QRS_NEXT_CUT()
PTP {E1 28976.874,E2 28976.874}
PTP {X 0,Y 607.926,A -85,B 0,C 180,E1 28976.874,E2 28976.874,E3 0,E4 0,E5 0,E6 0}
QRS_SPEED_INIT()
LIN {X 0,Y 607.926,Z 799,A -85,B 0,C 180,E1 28976.874,E2 28976.874,E3 0,E4 0,E5 0,E6 0} C_VEL
LIN {X 0,Y 607.926,Z 746.583,A -85,B 0,C 180,E1 28976.874,E2 28976.874} C_VEL
LIN {X 0,Y 607.926,Z 738.171,A -85,B 0,C 180,E1 28976.874,E2 28976.874} C_VEL
LIN {X 0,Y 607.916,Z 736.195,A -85,B 0,C 180,E1 28976.715,E2 28976.715} C_VEL
LIN {X 0,Y 607.917,Z 732.197,A -85,B 0,C 180,E1 28974.904,E2 28974.904} C_VEL
LIN {X 0,Y 607.91,Z 726.378,A -85,B 0,C 180,E1 28973.104,E2 28973.104} C_VEL
LIN {X 0,Y 607.913,Z 719.011,A -85,B 0,C 180,E1 28971.392,E2 28971.392} C_VEL
LIN {X 0,Y 607.912,Z 710.203,A -85,B 0,C 180,E1 28969.768,E2 28969.768} C_VEL
LIN {X 0,Y 607.913,Z 699.301,A -85,B 0,C 180,E1 28968.132,E2 28968.132} C_VEL
LIN {X 0,Y 607.913,Z 686.828,A -85,B 0,C 180,E1 28966.59,E2 28966.59} C_VEL
LIN {X 0,Y 607.915,Z 673.153,A -85,B 0,C 180,E1 28965.181,E2 28965.181} C_VEL
LIN {X 0,Y 607.917,Z 658.405,A -85,B 0,C 180,E1 28963.91,E2 28963.91} C_VEL
LIN {X 0,Y 607.919,Z 642.683,A -85,B 0,C 180,E1 28962.779,E2 28962.779} C_VEL
LIN {X 0,Y 607.913,Z 626.024,A -85,B 0,C 180,E1 28961.79,E2 28961.79} C_VEL
LIN {X 0,Y 607.915,Z 608.442,A -85,B 0,C 180,E1 28960.944,E2 28960.944} C_VEL
LIN {X 0,Y 607.91,Z 590.522,A -85,B 0,C 180,E1 28960.27,E2 28960.27} C_VEL
LIN {X 0,Y 607.91,Z 572.648,A -85,B 0,C 180,E1 28959.768,E2 28959.768} C_VEL
LIN {X 0,Y 607.915,Z 554.05,A -85,B 0,C 180,E1 28959.417,E2 28959.417} C_VEL
LIN {X 0,Y 607.913,Z 342.093,A -85,B 0,C 180,E1 28956.75,E2 28956.75} C_VEL
LIN {X 0,Y 607.872,Z 299.576,A -85,B 0,C 180,E1 28953.695,E2 28953.695} C_VEL
LIN {X 0,Y 607.918,Z 261.354,A -85,B 0,C 180,E1 28950.867,E2 28950.867} C_VEL
LIN {X 0,Y 607.912,Z 260.757,A -85,B 0,C 180,E1 28950.65,E2 28950.65} C_VEL
LIN {X 0,Y 607.867,Z 260.764,A -85,B 0,C 180,E1 28947.546,E2 28947.546} C_VEL
LIN {X 0,Y 607.884,Z 260.759,A -85,B 0,C 180,E1 28944.273,E2 28944.273} C_VEL
LIN {X 0,Y 607.911,Z 260.765,A -85,B 0,C 180,E1 28941.196,E2 28941.196} C_VEL
LIN {X 0,Y 607.881,Z 260.759,A -85,B 0,C 180,E1 28937.975,E2 28937.975} C_VEL
LIN {X 0,Y 607.906,Z 260.759,A -85,B 0,C 180,E1 28934.855,E2 28934.855} C_VEL
LIN {X 0,Y 607.896,Z 260.762,A -85,B 0,C 180,E1 28931.691,E2 28931.691} C_VEL
LIN {X 0,Y 607.919,Z 260.754,A -85,B 0,C 180,E1 28928.441,E2 28928.441} C_VEL
LIN {X 0,Y 607.897,Z 260.762,A -85,B 0,C 180,E1 28925.168,E2 28925.168} C_VEL
LIN {X 0,Y 607.907,Z 260.758,A -85,B 0,C 180,E1 28922.091,E2 28922.091} C_VEL
LIN {X 0,Y 607.882,Z 260.759,A -85,B 0,C 180,E1 28918.92,E2 28918.92} C_VEL
LIN {X 0,Y 607.913,Z 260.765,A -85,B 0,C 180,E1 28915.736,E2 28915.736} C_VEL
LIN {X 0,Y 607.88,Z 260.759,A -85,B 0,C 180,E1 28912.638,E2 28912.638} C_VEL
LIN {X 0,Y 607.875,Z 260.763,A -85,B 0,C 180,E1 28909.407,E2 28909.407} C_VEL
LIN {X 0,Y 607.886,Z 260.76,A -85,B 0,C 180,E1 28906.435,E2 28906.435} C_VEL
LIN {X 0,Y 607.853,Z 260.764,A -85,B 0,C 180,E1 28903.315,E2 28903.315} C_VEL
LIN {X 0,Y 607.88,Z 260.763,A -85,B 0,C 180,E1 28900.385,E2 28900.385} C_VEL
LIN {X 0,Y 607.835,Z 260.767,A -85,B 0,C 180,E1 28897.278,E2 28897.278} C_VEL
LIN {X 0,Y 607.89,Z 260.966,A -85,B 0,C 180,E1 28896.257,E2 28896.257} C_VEL
LIN {X 0,Y 607.917,Z 266.861,A -85,B 0,C 180,E1 28895.759,E2 28895.759} C_VEL
LIN {X 0,Y 607.901,Z 307.026,A -85,B 0,C 180,E1 28892.688,E2 28892.688} C_VEL
LIN {X 0,Y 607.906,Z 348.222,A -85,B 0,C 180,E1 28889.624,E2 28889.624} C_VEL
LIN {X 0,Y 607.895,Z 390.467,A -85,B 0,C 180,E1 28886.559,E2 28886.559} C_VEL
LIN {X 0,Y 607.879,Z 435.108,A -85,B 0,C 180,E1 28883.39,E2 28883.39} C_VEL
LIN {X 0,Y 607.906,Z 472.483,A -85,B 0,C 180,E1 28880.797,E2 28880.797} C_VEL
LIN {X 0,Y 607.898,Z 614.271,A -85,B 0,C 180,E1 28879.072,E2 28879.072} C_VEL
LIN {X 0,Y 607.919,Z 631.005,A -85,B 0,C 180,E1 28878.69,E2 28878.69} C_VEL
LIN {X 0,Y 607.916,Z 645.866,A -85,B 0,C 180,E1 28878.185,E2 28878.185} C_VEL
LIN {X 0,Y 607.916,Z 660.472,A -85,B 0,C 180,E1 28877.51,E2 28877.51} C_VEL
LIN {X 0,Y 607.918,Z 675.006,A -85,B 0,C 180,E1 28876.64,E2 28876.64} C_VEL
LIN {X 0,Y 607.918,Z 687.294,A -85,B 0,C 180,E1 28875.718,E2 28875.718} C_VEL
LIN {X 0,Y 607.918,Z 699.759,A -85,B 0,C 180,E1 28874.548,E2 28874.548} C_VEL
LIN {X 0,Y 607.917,Z 709.872,A -85,B 0,C 180,E1 28873.372,E2 28873.372} C_VEL
LIN {X 0,Y 607.917,Z 719.257,A -85,B 0,C 180,E1 28871.99,E2 28871.99} C_VEL
LIN {X 0,Y 607.917,Z 726.624,A -85,B 0,C 180,E1 28870.597,E2 28870.597} C_VEL
LIN {X 0,Y 607.918,Z 732.436,A -85,B 0,C 180,E1 28869.091,E2 28869.091} C_VEL
LIN {X 0,Y 607.919,Z 736.408,A -85,B 0,C 180,E1 28867.57,E2 28867.57} C_VEL
LIN {X 0,Y 607.917,Z 738.54,A -85,B 0,C 180,E1 28866.032,E2 28866.032} C_VEL
LIN {X 0,Y 607.916,Z 738.894,A -85,B 0,C 180,E1 28864.476,E2 28864.476} C_VEL
LIN {X 0,Y 607.914,Z 737.56,A -85,B 0,C 180,E1 28863.004,E2 28863.004} C_VEL
LIN {X 0,Y 607.916,Z 734.271,A -85,B 0,C 180,E1 28861.437,E2 28861.437} C_VEL
LIN {X 0,Y 607.914,Z 729.539,A -85,B 0,C 180,E1 28860.002,E2 28860.002} C_VEL
LIN {X 0,Y 607.915,Z 722.969,A -85,B 0,C 180,E1 28858.577,E2 28858.577} C_VEL
LIN {X 0,Y 607.919,Z 714.179,A -85,B 0,C 180,E1 28857.13,E2 28857.13} C_VEL
LIN {X 0,Y 607.917,Z 704.536,A -85,B 0,C 180,E1 28855.887,E2 28855.887} C_VEL
LIN {X 0,Y 607.918,Z 692.695,A -85,B 0,C 180,E1 28854.666,E2 28854.666} C_VEL
LIN {X 0,Y 607.918,Z 680.197,A -85,B 0,C 180,E1 28853.637,E2 28853.637} C_VEL
LIN {X 0,Y 607.906,Z 665.842,A -85,B 0,C 180,E1 28852.694,E2 28852.694} C_VEL
LIN {X 0,Y 607.904,Z 651.24,A -85,B 0,C 180,E1 28851.953,E2 28851.953} C_VEL
LIN {X 0,Y 607.917,Z 635.281,A -85,B 0,C 180,E1 28851.348,E2 28851.348} C_VEL
LIN {X 0,Y 607.896,Z 619.814,A -85,B 0,C 180,E1 28850.941,E2 28850.941} C_VEL
LIN {X 0,Y 607.871,Z 600.343,A -85,B 0,C 180,E1 28850.652,E2 28850.652} C_VEL
LIN {X 0,Y 607.901,Z 472.16,A -85,B 0,C 180,E1 28849.1,E2 28849.1} C_VEL
LIN {X 0,Y 607.844,Z 432.037,A -85,B 0,C 180,E1 28846.303,E2 28846.303} C_VEL
LIN {X 0,Y 607.882,Z 388.77,A -85,B 0,C 180,E1 28843.228,E2 28843.228} C_VEL
LIN {X 0,Y 607.899,Z 347.838,A -85,B 0,C 180,E1 28840.257,E2 28840.257} C_VEL
LIN {X 0,Y 607.913,Z 306.577,A -85,B 0,C 180,E1 28837.189,E2 28837.189} C_VEL
LIN {X 0,Y 607.919,Z 265.74,A -85,B 0,C 180,E1 28834.064,E2 28834.064} C_VEL
LIN {X 0,Y 607.913,Z 260.992,A -85,B 0,C 180,E1 28833.661,E2 28833.661} C_VEL
LIN {X 0,Y 607.864,Z 260.761,A -85,B 0,C 180,E1 28830.657,E2 28830.657} C_VEL
LIN {X 0,Y 607.915,Z 260.761,A -85,B 0,C 180,E1 28827.566,E2 28827.566} C_VEL
LIN {X 0,Y 607.864,Z 260.761,A -85,B 0,C 180,E1 28824.489,E2 28824.489} C_VEL
LIN {X 0,Y 607.915,Z 260.758,A -85,B 0,C 180,E1 28821.315,E2 28821.315} C_VEL
LIN {X 0,Y 607.871,Z 260.762,A -85,B 0,C 180,E1 28818.212,E2 28818.212} C_VEL
LIN {X 0,Y 607.895,Z 260.757,A -85,B 0,C 180,E1 28814.966,E2 28814.966} C_VEL
LIN {X 0,Y 607.892,Z 260.764,A -85,B 0,C 180,E1 28811.865,E2 28811.865} C_VEL
LIN {X 0,Y 607.874,Z 260.759,A -85,B 0,C 180,E1 28808.609,E2 28808.609} C_VEL
LIN {X 0,Y 607.911,Z 260.766,A -85,B 0,C 180,E1 28805.569,E2 28805.569} C_VEL
LIN {X 0,Y 607.871,Z 260.759,A -85,B 0,C 180,E1 28802.451,E2 28802.451} C_VEL
LIN {X 0,Y 607.914,Z 260.762,A -85,B 0,C 180,E1 28799.341,E2 28799.341} C_VEL
LIN {X 0,Y 607.87,Z 260.76,A -85,B 0,C 180,E1 28796.228,E2 28796.228} C_VEL
LIN {X 0,Y 607.911,Z 260.759,A -85,B 0,C 180,E1 28793.104,E2 28793.104} C_VEL
LIN {X 0,Y 607.872,Z 260.761,A -85,B 0,C 180,E1 28790.055,E2 28790.055} C_VEL
LIN {X 0,Y 607.915,Z 260.756,A -85,B 0,C 180,E1 28786.818,E2 28786.818} C_VEL
LIN {X 0,Y 607.89,Z 260.763,A -85,B 0,C 180,E1 28783.665,E2 28783.665} C_VEL
LIN {X 0,Y 607.882,Z 260.758,A -85,B 0,C 180,E1 28780.395,E2 28780.395} C_VEL
LIN {X 0,Y 607.916,Z 260.764,A -85,B 0,C 180,E1 28777.263,E2 28777.263} C_VEL
LIN {X 0,Y 607.875,Z 260.759,A -85,B 0,C 180,E1 28774.119,E2 28774.119} C_VEL
LIN {X 0,Y 607.911,Z 260.76,A -85,B 0,C 180,E1 28770.975,E2 28770.975} C_VEL
LIN {X 0,Y 607.875,Z 260.76,A -85,B 0,C 180,E1 28767.894,E2 28767.894} C_VEL
LIN {X 0,Y 607.914,Z 260.757,A -85,B 0,C 180,E1 28764.739,E2 28764.739} C_VEL
LIN {X 0,Y 607.88,Z 260.761,A -85,B 0,C 180,E1 28761.677,E2 28761.677} C_VEL
LIN {X 0,Y 607.905,Z 260.756,A -85,B 0,C 180,E1 28758.447,E2 28758.447} C_VEL
LIN {X 0,Y 607.908,Z 260.764,A -85,B 0,C 180,E1 28755.255,E2 28755.255} C_VEL
LIN {X 0,Y 607.882,Z 260.758,A -85,B 0,C 180,E1 28752.022,E2 28752.022} C_VEL
LIN {X 0,Y 607.912,Z 260.762,A -85,B 0,C 180,E1 28748.922,E2 28748.922} C_VEL
LIN {X 0,Y 607.878,Z 260.757,A -85,B 0,C 180,E1 28745.816,E2 28745.816} C_VEL
LIN {X 0,Y 607.909,Z 260.758,A -85,B 0,C 180,E1 28742.758,E2 28742.758} C_VEL
LIN {X 0,Y 607.901,Z 261.045,A -85,B 0,C 180,E1 28741.19,E2 28741.19} C_VEL
LIN {X 0,Y 607.917,Z 270.434,A -85,B 0,C 180,E1 28740.544,E2 28740.544} C_VEL
LIN {X 0,Y 607.883,Z 315.134,A -85,B 0,C 180,E1 28737.7,E2 28737.7} C_VEL
LIN {X 0,Y 607.916,Z 528.002,A -85,B 0,C 180,E1 28734.938,E2 28734.938} C_VEL
LIN {X 0,Y 607.917,Z 577.773,A -85,B 0,C 180,E1 28734.278,E2 28734.278} C_VEL
LIN {X 0,Y 607.906,Z 597.727,A -85,B 0,C 180,E1 28733.84,E2 28733.84} C_VEL
LIN {X 0,Y 607.911,Z 617.08,A -85,B 0,C 180,E1 28733.248,E2 28733.248} C_VEL
LIN {X 0,Y 607.916,Z 636.502,A -85,B 0,C 180,E1 28732.482,E2 28732.482} C_VEL
LIN {X 0,Y 607.919,Z 655.181,A -85,B 0,C 180,E1 28731.566,E2 28731.566} C_VEL
LIN {X 0,Y 607.917,Z 673.777,A -85,B 0,C 180,E1 28730.456,E2 28730.456} C_VEL
LIN {X 0,Y 607.915,Z 691.264,A -85,B 0,C 180,E1 28729.204,E2 28729.204} C_VEL
LIN {X 0,Y 607.914,Z 707.171,A -85,B 0,C 180,E1 28727.862,E2 28727.862} C_VEL
LIN {X 0,Y 607.917,Z 721.68,A -85,B 0,C 180,E1 28726.432,E2 28726.432} C_VEL
LIN {X 0,Y 607.909,Z 735.27,A -85,B 0,C 180,E1 28724.866,E2 28724.866} C_VEL
LIN {X 0,Y 607.906,Z 747.75,A -85,B 0,C 180,E1 28723.171,E2 28723.171} C_VEL
LIN {X 0,Y 607.905,Z 758.257,A -85,B 0,C 180,E1 28721.478,E2 28721.478} C_VEL
LIN {X 0,Y 607.912,Z 767.565,A -85,B 0,C 180,E1 28719.657,E2 28719.657} C_VEL
LIN {X 0,Y 607.914,Z 774.977,A -85,B 0,C 180,E1 28717.845,E2 28717.845} C_VEL
LIN {X 0,Y 607.918,Z 780.991,A -85,B 0,C 180,E1 28715.946,E2 28715.946} C_VEL
LIN {X 0,Y 607.916,Z 785.294,A -85,B 0,C 180,E1 28714.054,E2 28714.054} C_VEL
LIN {X 0,Y 607.914,Z 788.04,A -85,B 0,C 180,E1 28712.073,E2 28712.073} C_VEL
LIN {X 0,Y 607.912,Z 788.984,A -85,B 0,C 180,E1 28710.093,E2 28710.093} C_VEL
LIN {X 0,Y 607.91,Z 788.239,A -85,B 0,C 180,E1 28708.208,E2 28708.208} C_VEL
LIN {X 0,Y 607.915,Z 785.764,A -85,B 0,C 180,E1 28706.227,E2 28706.227} C_VEL
LIN {X 0,Y 607.914,Z 781.492,A -85,B 0,C 180,E1 28704.241,E2 28704.241} C_VEL
LIN {X 0,Y 607.913,Z 776.031,A -85,B 0,C 180,E1 28702.438,E2 28702.438} C_VEL
LIN {X 0,Y 607.911,Z 768.837,A -85,B 0,C 180,E1 28700.628,E2 28700.628} C_VEL
LIN {X 0,Y 607.909,Z 760.319,A -85,B 0,C 180,E1 28698.904,E2 28698.904} C_VEL
LIN {X 0,Y 607.914,Z 749.368,A -85,B 0,C 180,E1 28697.074,E2 28697.074} C_VEL
LIN {X 0,Y 607.911,Z 737.579,A -85,B 0,C 180,E1 28695.424,E2 28695.424} C_VEL
LIN {X 0,Y 607.918,Z 724.302,A -85,B 0,C 180,E1 28693.846,E2 28693.846} C_VEL
LIN {X 0,Y 607.916,Z 709.355,A -85,B 0,C 180,E1 28692.334,E2 28692.334} C_VEL
LIN {X 0,Y 607.914,Z 692.556,A -85,B 0,C 180,E1 28690.894,E2 28690.894} C_VEL
LIN {X 0,Y 607.916,Z 674.521,A -85,B 0,C 180,E1 28689.592,E2 28689.592} C_VEL
LIN {X 0,Y 607.919,Z 656.038,A -85,B 0,C 180,E1 28688.482,E2 28688.482} C_VEL
LIN {X 0,Y 607.916,Z 637.586,A -85,B 0,C 180,E1 28687.568,E2 28687.568} C_VEL
LIN {X 0,Y 607.909,Z 618.324,A -85,B 0,C 180,E1 28686.795,E2 28686.795} C_VEL
LIN {X 0,Y 607.906,Z 598.676,A -85,B 0,C 180,E1 28686.184,E2 28686.184} C_VEL
LIN {X 0,Y 607.918,Z 578.992,A -85,B 0,C 180,E1 28685.746,E2 28685.746} C_VEL
LIN {X 0,Y 607.91,Z 541.04,A -85,B 0,C 180,E1 28685.228,E2 28685.228} C_VEL
LIN {X 0,Y 607.883,Z 316.158,A -85,B 0,C 180,E1 28682.324,E2 28682.324} C_VEL
LIN {X 0,Y 607.885,Z 313.372,A -85,B 0,C 180,E1 28682.196,E2 28682.196} C_VEL
LIN {X 0,Y 607.918,Z 267.016,A -85,B 0,C 180,E1 28679.235,E2 28679.235} C_VEL
LIN {X 0,Y 607.903,Z 261.097,A -85,B 0,C 180,E1 28678.822,E2 28678.822} C_VEL
LIN {X 0,Y 607.884,Z 260.755,A -85,B 0,C 180,E1 28678.073,E2 28678.073} C_VEL
LIN {X 0,Y 607.904,Z 260.764,A -85,B 0,C 180,E1 28674.83,E2 28674.83} C_VEL
LIN {X 0,Y 607.919,Z 260.756,A -85,B 0,C 180,E1 28671.559,E2 28671.559} C_VEL
LIN {X 0,Y 607.873,Z 260.761,A -85,B 0,C 180,E1 28668.354,E2 28668.354} C_VEL
LIN {X 0,Y 607.913,Z 260.76,A -85,B 0,C 180,E1 28665.255,E2 28665.255} C_VEL
LIN {X 0,Y 607.868,Z 260.76,A -85,B 0,C 180,E1 28662.152,E2 28662.152} C_VEL
LIN {X 0,Y 607.917,Z 260.764,A -85,B 0,C 180,E1 28659.045,E2 28659.045} C_VEL
LIN {X 0,Y 607.867,Z 260.76,A -85,B 0,C 180,E1 28655.959,E2 28655.959} C_VEL
LIN {X 0,Y 607.894,Z 260.765,A -85,B 0,C 180,E1 28652.761,E2 28652.761} C_VEL
LIN {X 0,Y 607.875,Z 260.757,A -85,B 0,C 180,E1 28649.717,E2 28649.717} C_VEL
LIN {X 0,Y 607.917,Z 261.074,A -85,B 0,C 180,E1 28649.079,E2 28649.079} C_VEL
LIN {X 0,Y 607.882,Z 296.062,A -85,B 0,C 180,E1 28646.471,E2 28646.471} C_VEL
LIN {X 0,Y 607.915,Z 339.268,A -85,B 0,C 180,E1 28643.352,E2 28643.352} C_VEL
LIN {X 0,Y 607.913,Z 342.484,A -85,B 0,C 180,E1 28643.147,E2 28643.147} C_VEL
LIN {X 0,Y 607.914,Z 559.808,A -85,B 0,C 180,E1 28640.407,E2 28640.407} C_VEL
LIN {X 0,Y 607.914,Z 579.217,A -85,B 0,C 180,E1 28639.98,E2 28639.98} C_VEL
LIN {X 0,Y 607.914,Z 597.431,A -85,B 0,C 180,E1 28639.404,E2 28639.404} C_VEL
LIN {X 0,Y 607.915,Z 615.767,A -85,B 0,C 180,E1 28638.639,E2 28638.639} C_VEL
LIN {X 0,Y 607.918,Z 633.298,A -85,B 0,C 180,E1 28637.714,E2 28637.714} C_VEL
LIN {X 0,Y 607.915,Z 650.04,A -85,B 0,C 180,E1 28636.629,E2 28636.629} C_VEL
LIN {X 0,Y 607.917,Z 665.659,A -85,B 0,C 180,E1 28635.404,E2 28635.404} C_VEL
LIN {X 0,Y 607.915,Z 679.684,A -85,B 0,C 180,E1 28634.088,E2 28634.088} C_VEL
LIN {X 0,Y 607.915,Z 692.662,A -85,B 0,C 180,E1 28632.635,E2 28632.635} C_VEL
LIN {X 0,Y 607.917,Z 704.133,A -85,B 0,C 180,E1 28631.095,E2 28631.095} C_VEL
LIN {X 0,Y 607.911,Z 714.103,A -85,B 0,C 180,E1 28629.466,E2 28629.466} C_VEL
LIN {X 0,Y 607.912,Z 722.146,A -85,B 0,C 180,E1 28627.846,E2 28627.846} C_VEL
LIN {X 0,Y 607.91,Z 728.788,A -85,B 0,C 180,E1 28626.137,E2 28626.137} C_VEL
LIN {X 0,Y 607.905,Z 733.703,A -85,B 0,C 180,E1 28624.433,E2 28624.433} C_VEL
LIN {X 0,Y 607.908,Z 737.107,A -85,B 0,C 180,E1 28622.639,E2 28622.639} C_VEL
LIN {X 0,Y 607.917,Z 738.818,A -85,B 0,C 180,E1 28620.754,E2 28620.754} C_VEL
LIN {X 0,Y 607.915,Z 738.727,A -85,B 0,C 180,E1 28618.963,E2 28618.963} C_VEL
LIN {X 0,Y 607.912,Z 736.955,A -85,B 0,C 180,E1 28617.171,E2 28617.171} C_VEL
LIN {X 0,Y 607.916,Z 736.195,A -85,B 0,C 180,E1 28616.715,E2 28616.715} C_VEL
LIN {X 0,Y 606.897,Z 734.89,A -85,B 0,C 180,E1 28615.999,E2 28615.999} C_VEL
LIN {X 0,Y 601.771,Z 731.347,A -85,B 0,C 180,E1 28614.518,E2 28614.518} C_VEL
LIN {X 0,Y 600.007,Z 728.896,A -85,B 0,C 180,E1 28613.716,E2 28613.716} C_VEL
LIN {X 0,Y 599.918,Z 728.211,A -85,B 0,C 180,E1 28613.514,E2 28613.514} C_VEL
LIN {X 0,Y 599.921,Z 721.302,A -85,B 0,C 180,E1 28611.759,E2 28611.759} C_VEL
LIN {X 0,Y 599.942,Z 712.5,A -85,B 0,C 180,E1 28610.018,E2 28610.018} C_VEL
LIN {X 0,Y 599.964,Z 702.139,A -85,B 0,C 180,E1 28608.366,E2 28608.366} C_VEL
LIN {X 0,Y 600.005,Z 690.217,A -85,B 0,C 180,E1 28606.803,E2 28606.803} C_VEL
LIN {X 0,Y 600.044,Z 676.686,A -85,B 0,C 180,E1 28605.328,E2 28605.328} C_VEL
LIN {X 0,Y 600.096,Z 662.408,A -85,B 0,C 180,E1 28604.025,E2 28604.025} C_VEL
LIN {X 0,Y 600.153,Z 647.039,A -85,B 0,C 180,E1 28602.849,E2 28602.849} C_VEL
LIN {X 0,Y 600.218,Z 630.474,A -85,B 0,C 180,E1 28601.799,E2 28601.799} C_VEL
LIN {X 0,Y 600.273,Z 614.032,A -85,B 0,C 180,E1 28600.945,E2 28600.945} C_VEL
LIN {X 0,Y 600.329,Z 595.811,A -85,B 0,C 180,E1 28600.193,E2 28600.193} C_VEL
LIN {X 0,Y 600.38,Z 576.816,A -85,B 0,C 180,E1 28599.606,E2 28599.606} C_VEL
LIN {X 0,Y 600.415,Z 557.875,A -85,B 0,C 180,E1 28599.205,E2 28599.205} C_VEL
LIN {X 0,Y 600.429,Z 342.582,A -85,B 0,C 180,E1 28596.459,E2 28596.459} C_VEL
LIN {X 0,Y 600.422,Z 301.598,A -85,B 0,C 180,E1 28593.494,E2 28593.494} C_VEL
LIN {X 0,Y 600.567,Z 263.941,A -85,B 0,C 180,E1 28590.68,E2 28590.68} C_VEL
LIN {X 0,Y 599.967,Z 261.874,A -85,B 0,C 180,E1 28590.442,E2 28590.442} C_VEL
LIN {X 0,Y 599.936,Z 261.754,A -85,B 0,C 180,E1 28587.43,E2 28587.43} C_VEL
LIN {X 0,Y 599.94,Z 261.748,A -85,B 0,C 180,E1 28584.198,E2 28584.198} C_VEL
LIN {X 0,Y 599.974,Z 261.753,A -85,B 0,C 180,E1 28581.077,E2 28581.077} C_VEL
LIN {X 0,Y 599.942,Z 261.749,A -85,B 0,C 180,E1 28577.871,E2 28577.871} C_VEL
LIN {X 0,Y 599.97,Z 261.746,A -85,B 0,C 180,E1 28574.691,E2 28574.691} C_VEL
LIN {X 0,Y 599.975,Z 261.753,A -85,B 0,C 180,E1 28571.415,E2 28571.415} C_VEL
LIN {X 0,Y 599.961,Z 261.746,A -85,B 0,C 180,E1 28568.13,E2 28568.13} C_VEL
LIN {X 0,Y 599.953,Z 261.749,A -85,B 0,C 180,E1 28564.981,E2 28564.981} C_VEL
LIN {X 0,Y 599.97,Z 261.751,A -85,B 0,C 180,E1 28561.778,E2 28561.778} C_VEL
LIN {X 0,Y 599.958,Z 261.745,A -85,B 0,C 180,E1 28558.564,E2 28558.564} C_VEL
LIN {X 0,Y 599.942,Z 261.75,A -85,B 0,C 180,E1 28555.256,E2 28555.256} C_VEL
LIN {X 0,Y 599.977,Z 261.748,A -85,B 0,C 180,E1 28552.092,E2 28552.092} C_VEL
LIN {X 0,Y 599.922,Z 261.751,A -85,B 0,C 180,E1 28548.966,E2 28548.966} C_VEL
LIN {X 0,Y 599.972,Z 261.753,A -85,B 0,C 180,E1 28545.862,E2 28545.862} C_VEL
LIN {X 0,Y 599.911,Z 261.752,A -85,B 0,C 180,E1 28542.834,E2 28542.834} C_VEL
LIN {X 0,Y 599.922,Z 261.755,A -85,B 0,C 180,E1 28539.595,E2 28539.595} C_VEL
LIN {X 0,Y 599.905,Z 261.757,A -85,B 0,C 180,E1 28536.701,E2 28536.701} C_VEL
LIN {X 0,Y 599.985,Z 262.18,A -85,B 0,C 180,E1 28536.508,E2 28536.508} C_VEL
LIN {X 0,Y 600.494,Z 265.704,A -85,B 0,C 180,E1 28536.214,E2 28536.214} C_VEL
LIN {X 0,Y 600.557,Z 294.621,A -85,B 0,C 180,E1 28534.011,E2 28534.011} C_VEL
LIN {X 0,Y 600.422,Z 335.458,A -85,B 0,C 180,E1 28530.907,E2 28530.907} C_VEL
LIN {X 0,Y 600.294,Z 376.693,A -85,B 0,C 180,E1 28527.853,E2 28527.853} C_VEL
LIN {X 0,Y 600.211,Z 418.923,A -85,B 0,C 180,E1 28524.792,E2 28524.792} C_VEL
LIN {X 0,Y 600.106,Z 464.253,A -85,B 0,C 180,E1 28521.57,E2 28521.57} C_VEL
LIN {X 0,Y 600.166,Z 472.786,A -85,B 0,C 180,E1 28521.001,E2 28521.001} C_VEL
LIN {X 0,Y 600.135,Z 615.243,A -85,B 0,C 180,E1 28519.241,E2 28519.241} C_VEL
LIN {X 0,Y 600.133,Z 632.155,A -85,B 0,C 180,E1 28518.84,E2 28518.84} C_VEL
LIN {X 0,Y 600.099,Z 646.835,A -85,B 0,C 180,E1 28518.322,E2 28518.322} C_VEL
LIN {X 0,Y 600.061,Z 662.094,A -85,B 0,C 180,E1 28517.589,E2 28517.589} C_VEL
LIN {X 0,Y 600.029,Z 676.504,A -85,B 0,C 180,E1 28516.695,E2 28516.695} C_VEL
LIN {X 0,Y 599.994,Z 689.443,A -85,B 0,C 180,E1 28515.674,E2 28515.674} C_VEL
LIN {X 0,Y 599.968,Z 701.086,A -85,B 0,C 180,E1 28514.537,E2 28514.537} C_VEL
LIN {X 0,Y 599.945,Z 711.629,A -85,B 0,C 180,E1 28513.244,E2 28513.244} C_VEL
LIN {X 0,Y 599.933,Z 720.689,A -85,B 0,C 180,E1 28511.842,E2 28511.842} C_VEL
LIN {X 0,Y 599.919,Z 727.663,A -85,B 0,C 180,E1 28510.429,E2 28510.429} C_VEL
LIN {X 0,Y 599.915,Z 733.208,A -85,B 0,C 180,E1 28508.901,E2 28508.901} C_VEL
LIN {X 0,Y 599.914,Z 736.863,A -85,B 0,C 180,E1 28507.358,E2 28507.358} C_VEL
LIN {X 0,Y 599.916,Z 738.786,A -85,B 0,C 180,E1 28505.692,E2 28505.692} C_VEL
LIN {X 0,Y 599.914,Z 738.746,A -85,B 0,C 180,E1 28504.16,E2 28504.16} C_VEL
LIN {X 0,Y 599.915,Z 736.787,A -85,B 0,C 180,E1 28502.507,E2 28502.507} C_VEL
LIN {X 0,Y 599.915,Z 733.146,A -85,B 0,C 180,E1 28500.989,E2 28500.989} C_VEL
LIN {X 0,Y 599.922,Z 727.529,A -85,B 0,C 180,E1 28499.449,E2 28499.449} C_VEL
LIN {X 0,Y 599.931,Z 720.468,A -85,B 0,C 180,E1 28498.029,E2 28498.029} C_VEL
LIN {X 0,Y 599.944,Z 711.414,A -85,B 0,C 180,E1 28496.637,E2 28496.637} C_VEL
LIN {X 0,Y 599.969,Z 701.066,A -85,B 0,C 180,E1 28495.371,E2 28495.371} C_VEL
LIN {X 0,Y 599.994,Z 689.078,A -85,B 0,C 180,E1 28494.204,E2 28494.204} C_VEL
LIN {X 0,Y 600.031,Z 676.113,A -85,B 0,C 180,E1 28493.189,E2 28493.189} C_VEL
LIN {X 0,Y 600.058,Z 661.752,A -85,B 0,C 180,E1 28492.302,E2 28492.302} C_VEL
LIN {X 0,Y 600.086,Z 647.798,A -85,B 0,C 180,E1 28491.629,E2 28491.629} C_VEL
LIN {X 0,Y 600.132,Z 632.099,A -85,B 0,C 180,E1 28491.069,E2 28491.069} C_VEL
LIN {X 0,Y 600.123,Z 615.12,A -85,B 0,C 180,E1 28490.667,E2 28490.667} C_VEL
LIN {X 0,Y 600.114,Z 472.239,A -85,B 0,C 180,E1 28488.893,E2 28488.893} C_VEL
LIN {X 0,Y 600.13,Z 431.749,A -85,B 0,C 180,E1 28486.034,E2 28486.034} C_VEL
LIN {X 0,Y 600.243,Z 387.092,A -85,B 0,C 180,E1 28482.815,E2 28482.815} C_VEL
LIN {X 0,Y 600.39,Z 347.187,A -85,B 0,C 180,E1 28479.879,E2 28479.879} C_VEL
LIN {X 0,Y 600.534,Z 305.133,A -85,B 0,C 180,E1 28476.707,E2 28476.707} C_VEL
LIN {X 0,Y 600.531,Z 270.72,A -85,B 0,C 180,E1 28474.074,E2 28474.074} C_VEL
LIN {X 0,Y 600.134,Z 262.619,A -85,B 0,C 180,E1 28473.468,E2 28473.468} C_VEL
LIN {X 0,Y 599.97,Z 261.765,A -85,B 0,C 180,E1 28473.291,E2 28473.291} C_VEL
LIN {X 0,Y 599.935,Z 261.753,A -85,B 0,C 180,E1 28470.22,E2 28470.22} C_VEL
LIN {X 0,Y 599.94,Z 261.748,A -85,B 0,C 180,E1 28466.925,E2 28466.925} C_VEL
LIN {X 0,Y 599.972,Z 261.754,A -85,B 0,C 180,E1 28463.785,E2 28463.785} C_VEL
LIN {X 0,Y 599.929,Z 261.749,A -85,B 0,C 180,E1 28460.589,E2 28460.589} C_VEL
LIN {X 0,Y 599.976,Z 261.75,A -85,B 0,C 180,E1 28457.456,E2 28457.456} C_VEL
LIN {X 0,Y 599.928,Z 261.75,A -85,B 0,C 180,E1 28454.379,E2 28454.379} C_VEL
LIN {X 0,Y 599.975,Z 261.747,A -85,B 0,C 180,E1 28451.244,E2 28451.244} C_VEL
LIN {X 0,Y 599.933,Z 261.751,A -85,B 0,C 180,E1 28448.135,E2 28448.135} C_VEL
LIN {X 0,Y 599.959,Z 261.746,A -85,B 0,C 180,E1 28444.876,E2 28444.876} C_VEL
LIN {X 0,Y 599.959,Z 261.753,A -85,B 0,C 180,E1 28441.719,E2 28441.719} C_VEL
LIN {X 0,Y 599.935,Z 261.748,A -85,B 0,C 180,E1 28438.472,E2 28438.472} C_VEL
LIN {X 0,Y 599.975,Z 261.751,A -85,B 0,C 180,E1 28435.316,E2 28435.316} C_VEL
LIN {X 0,Y 599.931,Z 261.75,A -85,B 0,C 180,E1 28432.146,E2 28432.146} C_VEL
LIN {X 0,Y 599.976,Z 261.746,A -85,B 0,C 180,E1 28428.951,E2 28428.951} C_VEL
LIN {X 0,Y 599.942,Z 261.751,A -85,B 0,C 180,E1 28425.819,E2 28425.819} C_VEL
LIN {X 0,Y 599.952,Z 261.746,A -85,B 0,C 180,E1 28422.544,E2 28422.544} C_VEL
LIN {X 0,Y 599.978,Z 261.753,A -85,B 0,C 180,E1 28419.311,E2 28419.311} C_VEL
LIN {X 0,Y 599.935,Z 261.749,A -85,B 0,C 180,E1 28416.11,E2 28416.11} C_VEL
LIN {X 0,Y 599.973,Z 261.748,A -85,B 0,C 180,E1 28412.938,E2 28412.938} C_VEL
LIN {X 0,Y 599.94,Z 261.75,A -85,B 0,C 180,E1 28409.781,E2 28409.781} C_VEL
LIN {X 0,Y 599.969,Z 261.745,A -85,B 0,C 180,E1 28406.522,E2 28406.522} C_VEL
LIN {X 0,Y 599.975,Z 261.754,A -85,B 0,C 180,E1 28403.254,E2 28403.254} C_VEL
LIN {X 0,Y 599.94,Z 261.748,A -85,B 0,C 180,E1 28400.05,E2 28400.05} C_VEL
LIN {X 0,Y 599.972,Z 261.75,A -85,B 0,C 180,E1 28396.901,E2 28396.901} C_VEL
LIN {X 0,Y 599.939,Z 261.749,A -85,B 0,C 180,E1 28393.758,E2 28393.758} C_VEL
LIN {X 0,Y 599.974,Z 261.746,A -85,B 0,C 180,E1 28390.535,E2 28390.535} C_VEL
LIN {X 0,Y 599.954,Z 261.753,A -85,B 0,C 180,E1 28387.344,E2 28387.344} C_VEL
LIN {X 0,Y 599.951,Z 261.748,A -85,B 0,C 180,E1 28384.052,E2 28384.052} C_VEL
LIN {X 0,Y 599.976,Z 261.995,A -85,B 0,C 180,E1 28381.589,E2 28381.589} C_VEL
LIN {X 0,Y 600.75,Z 265.362,A -85,B 0,C 180,E1 28381.282,E2 28381.282} C_VEL
LIN {X 0,Y 600.583,Z 311.765,A -85,B 0,C 180,E1 28378.275,E2 28378.275} C_VEL
LIN {X 0,Y 600.704,Z 316.046,A -85,B 0,C 180,E1 28378.038,E2 28378.038} C_VEL
LIN {X 0,Y 600.667,Z 519.783,A -85,B 0,C 180,E1 28375.367,E2 28375.367} C_VEL
LIN {X 0,Y 600.61,Z 578.292,A -85,B 0,C 180,E1 28374.583,E2 28374.583} C_VEL
LIN {X 0,Y 600.557,Z 598.764,A -85,B 0,C 180,E1 28374.124,E2 28374.124} C_VEL
LIN {X 0,Y 600.499,Z 617.817,A -85,B 0,C 180,E1 28373.526,E2 28373.526} C_VEL
LIN {X 0,Y 600.425,Z 637.639,A -85,B 0,C 180,E1 28372.725,E2 28372.725} C_VEL
LIN {X 0,Y 600.349,Z 656.078,A -85,B 0,C 180,E1 28371.8,E2 28371.8} C_VEL
LIN {X 0,Y 600.277,Z 674.551,A -85,B 0,C 180,E1 28370.677,E2 28370.677} C_VEL
LIN {X 0,Y 600.197,Z 692.585,A -85,B 0,C 180,E1 28369.359,E2 28369.359} C_VEL
LIN {X 0,Y 600.123,Z 709.379,A -85,B 0,C 180,E1 28367.901,E2 28367.901} C_VEL
LIN {X 0,Y 600.064,Z 724.878,A -85,B 0,C 180,E1 28366.309,E2 28366.309} C_VEL
LIN {X 0,Y 600.007,Z 738.373,A -85,B 0,C 180,E1 28364.671,E2 28364.671} C_VEL
LIN {X 0,Y 599.972,Z 750.023,A -85,B 0,C 180,E1 28363,E2 28363} C_VEL
LIN {X 0,Y 599.945,Z 760.331,A -85,B 0,C 180,E1 28361.243,E2 28361.243} C_VEL
LIN {X 0,Y 599.925,Z 769.36,A -85,B 0,C 180,E1 28359.373,E2 28359.373} C_VEL
LIN {X 0,Y 599.92,Z 776.383,A -85,B 0,C 180,E1 28357.565,E2 28357.565} C_VEL
LIN {X 0,Y 599.913,Z 782.004,A -85,B 0,C 180,E1 28355.642,E2 28355.642} C_VEL
LIN {X 0,Y 599.912,Z 785.926,A -85,B 0,C 180,E1 28353.726,E2 28353.726} C_VEL
LIN {X 0,Y 599.906,Z 788.307,A -85,B 0,C 180,E1 28351.718,E2 28351.718} C_VEL
LIN {X 0,Y 599.907,Z 788.962,A -85,B 0,C 180,E1 28349.808,E2 28349.808} C_VEL
LIN {X 0,Y 599.91,Z 787.949,A -85,B 0,C 180,E1 28347.802,E2 28347.802} C_VEL
LIN {X 0,Y 599.909,Z 785.133,A -85,B 0,C 180,E1 28345.794,E2 28345.794} C_VEL
LIN {X 0,Y 599.919,Z 780.733,A -85,B 0,C 180,E1 28343.876,E2 28343.876} C_VEL
LIN {X 0,Y 599.923,Z 774.616,A -85,B 0,C 180,E1 28341.951,E2 28341.951} C_VEL
LIN {X 0,Y 599.934,Z 766.799,A -85,B 0,C 180,E1 28340.053,E2 28340.053} C_VEL
LIN {X 0,Y 599.943,Z 757.711,A -85,B 0,C 180,E1 28338.268,E2 28338.268} C_VEL
LIN {X 0,Y 599.974,Z 746.81,A -85,B 0,C 180,E1 28336.507,E2 28336.507} C_VEL
LIN {X 0,Y 600.019,Z 734.479,A -85,B 0,C 180,E1 28334.833,E2 28334.833} C_VEL
LIN {X 0,Y 600.065,Z 720.733,A -85,B 0,C 180,E1 28333.245,E2 28333.245} C_VEL
LIN {X 0,Y 600.133,Z 705.441,A -85,B 0,C 180,E1 28331.741,E2 28331.741} C_VEL
LIN {X 0,Y 600.207,Z 688.595,A -85,B 0,C 180,E1 28330.335,E2 28330.335} C_VEL
LIN {X 0,Y 600.29,Z 671.337,A -85,B 0,C 180,E1 28329.117,E2 28329.117} C_VEL
LIN {X 0,Y 600.374,Z 653.234,A -85,B 0,C 180,E1 28328.044,E2 28328.044} C_VEL
LIN {X 0,Y 600.442,Z 634.219,A -85,B 0,C 180,E1 28327.118,E2 28327.118} C_VEL
LIN {X 0,Y 600.507,Z 614.815,A -85,B 0,C 180,E1 28326.368,E2 28326.368} C_VEL
LIN {X 0,Y 600.564,Z 594.781,A -85,B 0,C 180,E1 28325.776,E2 28325.776} C_VEL
LIN {X 0,Y 600.619,Z 574.279,A -85,B 0,C 180,E1 28325.354,E2 28325.354} C_VEL
LIN {X 0,Y 600.788,Z 328.828,A -85,B 0,C 180,E1 28322.137,E2 28322.137} C_VEL
LIN {X 0,Y 600.615,Z 315.45,A -85,B 0,C 180,E1 28321.946,E2 28321.946} C_VEL
LIN {X 0,Y 600.741,Z 269.622,A -85,B 0,C 180,E1 28318.998,E2 28318.998} C_VEL
LIN {X 0,Y 600.68,Z 264.235,A -85,B 0,C 180,E1 28318.639,E2 28318.639} C_VEL
LIN {X 0,Y 599.96,Z 261.887,A -85,B 0,C 180,E1 28318.386,E2 28318.386} C_VEL
LIN {X 0,Y 599.971,Z 261.752,A -85,B 0,C 180,E1 28315.244,E2 28315.244} C_VEL
LIN {X 0,Y 599.936,Z 261.749,A -85,B 0,C 180,E1 28312.17,E2 28312.17} C_VEL
LIN {X 0,Y 599.977,Z 261.754,A -85,B 0,C 180,E1 28308.958,E2 28308.958} C_VEL
LIN {X 0,Y 599.952,Z 261.747,A -85,B 0,C 180,E1 28305.776,E2 28305.776} C_VEL
LIN {X 0,Y 599.94,Z 261.752,A -85,B 0,C 180,E1 28302.554,E2 28302.554} C_VEL
LIN {X 0,Y 599.979,Z 261.747,A -85,B 0,C 180,E1 28299.415,E2 28299.415} C_VEL
LIN {X 0,Y 599.925,Z 261.751,A -85,B 0,C 180,E1 28296.229,E2 28296.229} C_VEL
LIN {X 0,Y 599.976,Z 261.752,A -85,B 0,C 180,E1 28293.135,E2 28293.135} C_VEL
LIN {X 0,Y 599.919,Z 261.744,A -85,B 0,C 180,E1 28290.11,E2 28290.11} C_VEL
LIN {X 0,Y 600.003,Z 262.027,A -85,B 0,C 180,E1 28289.43,E2 28289.43} C_VEL
LIN {X 0,Y 600.581,Z 265.108,A -85,B 0,C 180,E1 28289.141,E2 28289.141} C_VEL
LIN {X 0,Y 600.412,Z 305.124,A -85,B 0,C 180,E1 28286.156,E2 28286.156} C_VEL
LIN {X 0,Y 600.434,Z 342.643,A -85,B 0,C 180,E1 28283.45,E2 28283.45} C_VEL
LIN {X 0,Y 600.428,Z 548.25,A -85,B 0,C 180,E1 28280.843,E2 28280.843} C_VEL
LIN {X 0,Y 600.396,Z 568.16,A -85,B 0,C 180,E1 28280.511,E2 28280.511} C_VEL
LIN {X 0,Y 600.352,Z 587.649,A -85,B 0,C 180,E1 28279.994,E2 28279.994} C_VEL
LIN {X 0,Y 600.302,Z 605.96,A -85,B 0,C 180,E1 28279.324,E2 28279.324} C_VEL
LIN {X 0,Y 600.238,Z 623.416,A -85,B 0,C 180,E1 28278.501,E2 28278.501} C_VEL
LIN {X 0,Y 600.182,Z 640.833,A -85,B 0,C 180,E1 28277.482,E2 28277.482} C_VEL
LIN {X 0,Y 600.119,Z 657.022,A -85,B 0,C 180,E1 28276.326,E2 28276.326} C_VEL
LIN {X 0,Y 600.056,Z 672.23,A -85,B 0,C 180,E1 28275.017,E2 28275.017} C_VEL
LIN {X 0,Y 600.01,Z 686.053,A -85,B 0,C 180,E1 28273.589,E2 28273.589} C_VEL
LIN {X 0,Y 599.971,Z 697.976,A -85,B 0,C 180,E1 28272.121,E2 28272.121} C_VEL
LIN {X 0,Y 599.948,Z 708.519,A -85,B 0,C 180,E1 28270.563,E2 28270.563} C_VEL
LIN {X 0,Y 599.93,Z 717.663,A -85,B 0,C 180,E1 28268.916,E2 28268.916} C_VEL
LIN {X 0,Y 599.921,Z 725.343,A -85,B 0,C 180,E1 28267.18,E2 28267.18} C_VEL
LIN {X 0,Y 599.916,Z 731.456,A -85,B 0,C 180,E1 28265.355,E2 28265.355} C_VEL
LIN {X 0,Y 599.905,Z 735.71,A -85,B 0,C 180,E1 28263.535,E2 28263.535} C_VEL
LIN {X 0,Y 599.908,Z 738.196,A -85,B 0,C 180,E1 28261.719,E2 28261.719} C_VEL
LIN {X 0,Y 599.916,Z 738.994,A -85,B 0,C 180,E1 28259.904,E2 28259.904} C_VEL
LIN {X 0,Y 599.905,Z 738.107,A -85,B 0,C 180,E1 28258.089,E2 28258.089} C_VEL
LIN {X 0,Y 599.906,Z 735.523,A -85,B 0,C 180,E1 28256.273,E2 28256.273} C_VEL
LIN {X 0,Y 599.915,Z 731.175,A -85,B 0,C 180,E1 28254.452,E2 28254.452} C_VEL
LIN {X 0,Y 599.918,Z 728.211,A -85,B 0,C 180,E1 28253.514,E2 28253.514} C_VEL
LIN {X 0,Y 598.938,Z 725.736,A -85,B 0,C 180,E1 28252.817,E2 28252.817} C_VEL
LIN {X 0,Y 593.523,Z 719.553,A -85,B 0,C 180,E1 28251.285,E2 28251.285} C_VEL
LIN {X 0,Y 592.055,Z 716.348,A -85,B 0,C 180,E1 28250.612,E2 28250.612} C_VEL
LIN {X 0,Y 591.958,Z 715.339,A -85,B 0,C 180,E1 28250.419,E2 28250.419} C_VEL
LIN {X 0,Y 592.005,Z 705.364,A -85,B 0,C 180,E1 28248.701,E2 28248.701} C_VEL
LIN {X 0,Y 592.062,Z 694.15,A -85,B 0,C 180,E1 28247.119,E2 28247.119} C_VEL
LIN {X 0,Y 592.143,Z 681.452,A -85,B 0,C 180,E1 28245.628,E2 28245.628} C_VEL
LIN {X 0,Y 592.239,Z 667.137,A -85,B 0,C 180,E1 28244.221,E2 28244.221} C_VEL
LIN {X 0,Y 592.355,Z 651.963,A -85,B 0,C 180,E1 28242.976,E2 28242.976} C_VEL
LIN {X 0,Y 592.48,Z 635.562,A -85,B 0,C 180,E1 28241.858,E2 28241.858} C_VEL
LIN {X 0,Y 592.607,Z 617.997,A -85,B 0,C 180,E1 28240.882,E2 28240.882} C_VEL
LIN {X 0,Y 592.718,Z 601,A -85,B 0,C 180,E1 28240.128,E2 28240.128} C_VEL
LIN {X 0,Y 592.828,Z 582.281,A -85,B 0,C 180,E1 28239.488,E2 28239.488} C_VEL
LIN {X 0,Y 592.904,Z 563.275,A -85,B 0,C 180,E1 28239.029,E2 28239.029} C_VEL
LIN {X 0,Y 592.969,Z 536.355,A -85,B 0,C 180,E1 28238.64,E2 28238.64} C_VEL
LIN {X 0,Y 593.065,Z 343.72,A -85,B 0,C 180,E1 28236.169,E2 28236.169} C_VEL
LIN {X 0,Y 592.812,Z 341.522,A -85,B 0,C 180,E1 28236.087,E2 28236.087} C_VEL
LIN {X 0,Y 593.02,Z 299.426,A -85,B 0,C 180,E1 28232.974,E2 28232.974} C_VEL
LIN {X 0,Y 593.26,Z 266.996,A -85,B 0,C 180,E1 28230.519,E2 28230.519} C_VEL
LIN {X 0,Y 592.003,Z 262.881,A -85,B 0,C 180,E1 28230.088,E2 28230.088} C_VEL
LIN {X 0,Y 592.031,Z 262.736,A -85,B 0,C 180,E1 28227.056,E2 28227.056} C_VEL
LIN {X 0,Y 591.991,Z 262.739,A -85,B 0,C 180,E1 28223.881,E2 28223.881} C_VEL
LIN {X 0,Y 592.037,Z 262.736,A -85,B 0,C 180,E1 28220.704,E2 28220.704} C_VEL
LIN {X 0,Y 592.022,Z 262.741,A -85,B 0,C 180,E1 28217.423,E2 28217.423} C_VEL
LIN {X 0,Y 592.016,Z 262.736,A -85,B 0,C 180,E1 28214.127,E2 28214.127} C_VEL
LIN {X 0,Y 592.024,Z 262.738,A -85,B 0,C 180,E1 28210.942,E2 28210.942} C_VEL
LIN {X 0,Y 592.021,Z 262.739,A -85,B 0,C 180,E1 28207.776,E2 28207.776} C_VEL
LIN {X 0,Y 592.025,Z 262.734,A -85,B 0,C 180,E1 28204.574,E2 28204.574} C_VEL
LIN {X 0,Y 592.015,Z 262.74,A -85,B 0,C 180,E1 28201.232,E2 28201.232} C_VEL
LIN {X 0,Y 592.033,Z 262.737,A -85,B 0,C 180,E1 28198.003,E2 28198.003} C_VEL
LIN {X 0,Y 591.998,Z 262.737,A -85,B 0,C 180,E1 28194.87,E2 28194.87} C_VEL
LIN {X 0,Y 592.032,Z 262.741,A -85,B 0,C 180,E1 28191.708,E2 28191.708} C_VEL
LIN {X 0,Y 592.006,Z 262.738,A -85,B 0,C 180,E1 28188.514,E2 28188.514} C_VEL
LIN {X 0,Y 591.979,Z 262.739,A -85,B 0,C 180,E1 28185.278,E2 28185.278} C_VEL
LIN {X 0,Y 592.028,Z 262.74,A -85,B 0,C 180,E1 28182.188,E2 28182.188} C_VEL
LIN {X 0,Y 591.958,Z 262.745,A -85,B 0,C 180,E1 28179.137,E2 28179.137} C_VEL
LIN {X 0,Y 591.993,Z 262.99,A -85,B 0,C 180,E1 28176.827,E2 28176.827} C_VEL
LIN {X 0,Y 593.004,Z 267.28,A -85,B 0,C 180,E1 28176.439,E2 28176.439} C_VEL
LIN {X 0,Y 593.163,Z 305.254,A -85,B 0,C 180,E1 28173.577,E2 28173.577} C_VEL
LIN {X 0,Y 592.909,Z 347.591,A -85,B 0,C 180,E1 28170.339,E2 28170.339} C_VEL
LIN {X 0,Y 592.643,Z 388.451,A -85,B 0,C 180,E1 28167.293,E2 28167.293} C_VEL
LIN {X 0,Y 592.468,Z 432.944,A -85,B 0,C 180,E1 28164.044,E2 28164.044} C_VEL
LIN {X 0,Y 592.369,Z 472.692,A -85,B 0,C 180,E1 28161.219,E2 28161.219} C_VEL
LIN {X 0,Y 592.377,Z 615.341,A -85,B 0,C 180,E1 28159.43,E2 28159.43} C_VEL
LIN {X 0,Y 592.353,Z 632.233,A -85,B 0,C 180,E1 28159.024,E2 28159.024} C_VEL
LIN {X 0,Y 592.279,Z 648.091,A -85,B 0,C 180,E1 28158.447,E2 28158.447} C_VEL
LIN {X 0,Y 592.206,Z 663.716,A -85,B 0,C 180,E1 28157.669,E2 28157.669} C_VEL
LIN {X 0,Y 592.135,Z 677.581,A -85,B 0,C 180,E1 28156.775,E2 28156.775} C_VEL
LIN {X 0,Y 592.069,Z 691.026,A -85,B 0,C 180,E1 28155.677,E2 28155.677} C_VEL
LIN {X 0,Y 592.013,Z 702.334,A -85,B 0,C 180,E1 28154.524,E2 28154.524} C_VEL
LIN {X 0,Y 591.971,Z 712.659,A -85,B 0,C 180,E1 28153.214,E2 28153.214} C_VEL
LIN {X 0,Y 591.946,Z 720.917,A -85,B 0,C 180,E1 28151.894,E2 28151.894} C_VEL
LIN {X 0,Y 591.924,Z 727.836,A -85,B 0,C 180,E1 28150.462,E2 28150.462} C_VEL
LIN {X 0,Y 591.917,Z 733.333,A -85,B 0,C 180,E1 28148.914,E2 28148.914} C_VEL
LIN {X 0,Y 591.914,Z 736.929,A -85,B 0,C 180,E1 28147.349,E2 28147.349} C_VEL
LIN {X 0,Y 591.917,Z 738.742,A -85,B 0,C 180,E1 28145.767,E2 28145.767} C_VEL
LIN {X 0,Y 591.914,Z 738.784,A -85,B 0,C 180,E1 28144.204,E2 28144.204} C_VEL
LIN {X 0,Y 591.915,Z 736.894,A -85,B 0,C 180,E1 28142.54,E2 28142.54} C_VEL
LIN {X 0,Y 591.917,Z 733.353,A -85,B 0,C 180,E1 28141.002,E2 28141.002} C_VEL
LIN {X 0,Y 591.927,Z 727.81,A -85,B 0,C 180,E1 28139.442,E2 28139.442} C_VEL
LIN {X 0,Y 591.946,Z 720.667,A -85,B 0,C 180,E1 28137.971,E2 28137.971} C_VEL
LIN {X 0,Y 591.974,Z 711.62,A -85,B 0,C 180,E1 28136.552,E2 28136.552} C_VEL
LIN {X 0,Y 592.019,Z 701.684,A -85,B 0,C 180,E1 28135.31,E2 28135.31} C_VEL
LIN {X 0,Y 592.072,Z 689.863,A -85,B 0,C 180,E1 28134.129,E2 28134.129} C_VEL
LIN {X 0,Y 592.138,Z 677.349,A -85,B 0,C 180,E1 28133.118,E2 28133.118} C_VEL
LIN {X 0,Y 592.203,Z 663.732,A -85,B 0,C 180,E1 28132.242,E2 28132.242} C_VEL
LIN {X 0,Y 592.271,Z 648.277,A -85,B 0,C 180,E1 28131.471,E2 28131.471} C_VEL
LIN {X 0,Y 592.352,Z 632.347,A -85,B 0,C 180,E1 28130.89,E2 28130.89} C_VEL
LIN {X 0,Y 592.365,Z 615.505,A -85,B 0,C 180,E1 28130.482,E2 28130.482} C_VEL
LIN {X 0,Y 592.453,Z 528.737,A -85,B 0,C 180,E1 28129.391,E2 28129.391} C_VEL
LIN {X 0,Y 592.327,Z 472.394,A -85,B 0,C 180,E1 28128.683,E2 28128.683} C_VEL
LIN {X 0,Y 592.424,Z 432.221,A -85,B 0,C 180,E1 28125.812,E2 28125.812} C_VEL
LIN {X 0,Y 592.635,Z 386.909,A -85,B 0,C 180,E1 28122.502,E2 28122.502} C_VEL
LIN {X 0,Y 592.897,Z 347.818,A -85,B 0,C 180,E1 28119.587,E2 28119.587} C_VEL
LIN {X 0,Y 593.165,Z 306.048,A -85,B 0,C 180,E1 28116.395,E2 28116.395} C_VEL
LIN {X 0,Y 592.968,Z 269.99,A -85,B 0,C 180,E1 28113.695,E2 28113.695} C_VEL
LIN {X 0,Y 592.591,Z 264.884,A -85,B 0,C 180,E1 28113.313,E2 28113.313} C_VEL
LIN {X 0,Y 592.038,Z 262.941,A -85,B 0,C 180,E1 28113.109,E2 28113.109} C_VEL
LIN {X 0,Y 592.004,Z 262.744,A -85,B 0,C 180,E1 28110.107,E2 28110.107} C_VEL
LIN {X 0,Y 591.995,Z 262.738,A -85,B 0,C 180,E1 28106.805,E2 28106.805} C_VEL
LIN {X 0,Y 592.038,Z 262.742,A -85,B 0,C 180,E1 28103.7,E2 28103.7} C_VEL
LIN {X 0,Y 591.989,Z 262.738,A -85,B 0,C 180,E1 28100.568,E2 28100.568} C_VEL
LIN {X 0,Y 592.037,Z 262.738,A -85,B 0,C 180,E1 28097.393,E2 28097.393} C_VEL
LIN {X 0,Y 591.994,Z 262.74,A -85,B 0,C 180,E1 28094.202,E2 28094.202} C_VEL
LIN {X 0,Y 592.017,Z 262.735,A -85,B 0,C 180,E1 28090.904,E2 28090.904} C_VEL
LIN {X 0,Y 592.032,Z 262.742,A -85,B 0,C 180,E1 28087.668,E2 28087.668} C_VEL
LIN {X 0,Y 591.993,Z 262.738,A -85,B 0,C 180,E1 28084.456,E2 28084.456} C_VEL
LIN {X 0,Y 592.037,Z 262.738,A -85,B 0,C 180,E1 28081.258,E2 28081.258} C_VEL
LIN {X 0,Y 591.993,Z 262.739,A -85,B 0,C 180,E1 28078.161,E2 28078.161} C_VEL
LIN {X 0,Y 592.037,Z 262.735,A -85,B 0,C 180,E1 28074.962,E2 28074.962} C_VEL
LIN {X 0,Y 592.009,Z 262.741,A -85,B 0,C 180,E1 28071.747,E2 28071.747} C_VEL
LIN {X 0,Y 592.006,Z 262.736,A -85,B 0,C 180,E1 28068.505,E2 28068.505} C_VEL
LIN {X 0,Y 592.039,Z 262.741,A -85,B 0,C 180,E1 28065.326,E2 28065.326} C_VEL
LIN {X 0,Y 591.995,Z 262.738,A -85,B 0,C 180,E1 28062.098,E2 28062.098} C_VEL
LIN {X 0,Y 592.037,Z 262.735,A -85,B 0,C 180,E1 28058.917,E2 28058.917} C_VEL
LIN {X 0,Y 592.003,Z 262.74,A -85,B 0,C 180,E1 28055.77,E2 28055.77} C_VEL
LIN {X 0,Y 592.014,Z 262.735,A -85,B 0,C 180,E1 28052.435,E2 28052.435} C_VEL
LIN {X 0,Y 592.04,Z 262.742,A -85,B 0,C 180,E1 28049.222,E2 28049.222} C_VEL
LIN {X 0,Y 591.999,Z 262.737,A -85,B 0,C 180,E1 28046.011,E2 28046.011} C_VEL
LIN {X 0,Y 592.034,Z 262.737,A -85,B 0,C 180,E1 28042.855,E2 28042.855} C_VEL
LIN {X 0,Y 592.002,Z 262.739,A -85,B 0,C 180,E1 28039.695,E2 28039.695} C_VEL
LIN {X 0,Y 592.03,Z 262.734,A -85,B 0,C 180,E1 28036.427,E2 28036.427} C_VEL
LIN {X 0,Y 592.037,Z 262.743,A -85,B 0,C 180,E1 28033.149,E2 28033.149} C_VEL
LIN {X 0,Y 592.002,Z 262.737,A -85,B 0,C 180,E1 28029.924,E2 28029.924} C_VEL
LIN {X 0,Y 592.031,Z 262.732,A -85,B 0,C 180,E1 28026.821,E2 28026.821} C_VEL
LIN {X 0,Y 592.003,Z 262.742,A -85,B 0,C 180,E1 28023.629,E2 28023.629} C_VEL
LIN {X 0,Y 592.046,Z 262.985,A -85,B 0,C 180,E1 28021.995,E2 28021.995} C_VEL
LIN {X 0,Y 593.599,Z 267.831,A -85,B 0,C 180,E1 28021.537,E2 28021.537} C_VEL
LIN {X 0,Y 593.279,Z 314.401,A -85,B 0,C 180,E1 28018.484,E2 28018.484} C_VEL
LIN {X 0,Y 593.728,Z 318.555,A -85,B 0,C 180,E1 28018.362,E2 28018.362} C_VEL
LIN {X 0,Y 593.386,Z 547.087,A -85,B 0,C 180,E1 28015.342,E2 28015.342} C_VEL
LIN {X 0,Y 593.313,Z 579.752,A -85,B 0,C 180,E1 28014.875,E2 28014.875} C_VEL
LIN {X 0,Y 593.22,Z 600.256,A -85,B 0,C 180,E1 28014.403,E2 28014.403} C_VEL
LIN {X 0,Y 593.093,Z 620.024,A -85,B 0,C 180,E1 28013.759,E2 28013.759} C_VEL
LIN {X 0,Y 592.946,Z 638.839,A -85,B 0,C 180,E1 28012.972,E2 28012.972} C_VEL
LIN {X 0,Y 592.782,Z 657.865,A -85,B 0,C 180,E1 28011.989,E2 28011.989} C_VEL
LIN {X 0,Y 592.626,Z 676.018,A -85,B 0,C 180,E1 28010.853,E2 28010.853} C_VEL
LIN {X 0,Y 592.481,Z 693.207,A -85,B 0,C 180,E1 28009.57,E2 28009.57} C_VEL
LIN {X 0,Y 592.335,Z 709.911,A -85,B 0,C 180,E1 28008.093,E2 28008.093} C_VEL
LIN {X 0,Y 592.21,Z 725.363,A -85,B 0,C 180,E1 28006.476,E2 28006.476} C_VEL
LIN {X 0,Y 592.103,Z 739.141,A -85,B 0,C 180,E1 28004.772,E2 28004.772} C_VEL
LIN {X 0,Y 592.03,Z 751.335,A -85,B 0,C 180,E1 28002.974,E2 28002.974} C_VEL
LIN {X 0,Y 591.975,Z 761.369,A -85,B 0,C 180,E1 28001.199,E2 28001.199} C_VEL
LIN {X 0,Y 591.936,Z 770.066,A -85,B 0,C 180,E1 27999.331,E2 27999.331} C_VEL
LIN {X 0,Y 591.917,Z 777.052,A -85,B 0,C 180,E1 27997.454,E2 27997.454} C_VEL
LIN {X 0,Y 591.909,Z 782.51,A -85,B 0,C 180,E1 27995.524,E2 27995.524} C_VEL
LIN {X 0,Y 591.904,Z 786.242,A -85,B 0,C 180,E1 27993.582,E2 27993.582} C_VEL
LIN {X 0,Y 591.903,Z 788.374,A -85,B 0,C 180,E1 27991.645,E2 27991.645} C_VEL
LIN {X 0,Y 591.9,Z 788.917,A -85,B 0,C 180,E1 27989.612,E2 27989.612} C_VEL
LIN {X 0,Y 591.905,Z 787.838,A -85,B 0,C 180,E1 27987.675,E2 27987.675} C_VEL
LIN {X 0,Y 591.908,Z 784.971,A -85,B 0,C 180,E1 27985.639,E2 27985.639} C_VEL
LIN {X 0,Y 591.918,Z 780.48,A -85,B 0,C 180,E1 27983.695,E2 27983.695} C_VEL
LIN {X 0,Y 591.934,Z 774.262,A -85,B 0,C 180,E1 27981.744,E2 27981.744} C_VEL
LIN {X 0,Y 591.96,Z 766.172,A -85,B 0,C 180,E1 27979.784,E2 27979.784} C_VEL
LIN {X 0,Y 592.001,Z 756.562,A -85,B 0,C 180,E1 27977.91,E2 27977.91} C_VEL
LIN {X 0,Y 592.068,Z 745.492,A -85,B 0,C 180,E1 27976.124,E2 27976.124} C_VEL
LIN {X 0,Y 592.143,Z 732.929,A -85,B 0,C 180,E1 27974.425,E2 27974.425} C_VEL
LIN {X 0,Y 592.249,Z 718.879,A -85,B 0,C 180,E1 27972.815,E2 27972.815} C_VEL
LIN {X 0,Y 592.37,Z 703.835,A -85,B 0,C 180,E1 27971.345,E2 27971.345} C_VEL
LIN {X 0,Y 592.518,Z 687.276,A -85,B 0,C 180,E1 27969.966,E2 27969.966} C_VEL
LIN {X 0,Y 592.682,Z 669.735,A -85,B 0,C 180,E1 27968.733,E2 27968.733} C_VEL
LIN {X 0,Y 592.85,Z 651.248,A -85,B 0,C 180,E1 27967.646,E2 27967.646} C_VEL
LIN {X 0,Y 593.009,Z 632.397,A -85,B 0,C 180,E1 27966.735,E2 27966.735} C_VEL
LIN {X 0,Y 593.136,Z 612.748,A -85,B 0,C 180,E1 27965.982,E2 27965.982} C_VEL
LIN {X 0,Y 593.246,Z 592.965,A -85,B 0,C 180,E1 27965.412,E2 27965.412} C_VEL
LIN {X 0,Y 593.342,Z 572.319,A -85,B 0,C 180,E1 27965,E2 27965} C_VEL
LIN {X 0,Y 593.712,Z 329.973,A -85,B 0,C 180,E1 27961.791,E2 27961.791} C_VEL
LIN {X 0,Y 593.498,Z 316.574,A -85,B 0,C 180,E1 27961.6,E2 27961.6} C_VEL
LIN {X 0,Y 593.277,Z 314.36,A -85,B 0,C 180,E1 27961.513,E2 27961.513} C_VEL
LIN {X 0,Y 593.6,Z 267.671,A -85,B 0,C 180,E1 27958.452,E2 27958.452} C_VEL
LIN {X 0,Y 592.041,Z 262.954,A -85,B 0,C 180,E1 27958.002,E2 27958.002} C_VEL
LIN {X 0,Y 592.027,Z 262.744,A -85,B 0,C 180,E1 27954.827,E2 27954.827} C_VEL
LIN {X 0,Y 592.039,Z 262.735,A -85,B 0,C 180,E1 27951.574,E2 27951.574} C_VEL
LIN {X 0,Y 591.998,Z 262.74,A -85,B 0,C 180,E1 27948.412,E2 27948.412} C_VEL
LIN {X 0,Y 592.036,Z 262.739,A -85,B 0,C 180,E1 27945.23,E2 27945.23} C_VEL
LIN {X 0,Y 591.991,Z 262.739,A -85,B 0,C 180,E1 27942.107,E2 27942.107} C_VEL
LIN {X 0,Y 592.028,Z 262.744,A -85,B 0,C 180,E1 27938.869,E2 27938.869} C_VEL
LIN {X 0,Y 592,Z 262.739,A -85,B 0,C 180,E1 27935.759,E2 27935.759} C_VEL
LIN {X 0,Y 591.994,Z 262.744,A -85,B 0,C 180,E1 27932.486,E2 27932.486} C_VEL
LIN {X 0,Y 592.025,Z 262.972,A -85,B 0,C 180,E1 27929.798,E2 27929.798} C_VEL
LIN {X 0,Y 593.256,Z 267.278,A -85,B 0,C 180,E1 27929.369,E2 27929.369} C_VEL
LIN {X 0,Y 592.959,Z 307.602,A -85,B 0,C 180,E1 27926.326,E2 27926.326} C_VEL
LIN {X 0,Y 592.881,Z 342.554,A -85,B 0,C 180,E1 27923.769,E2 27923.769} C_VEL
LIN {X 0,Y 593.208,Z 348.346,A -85,B 0,C 180,E1 27923.675,E2 27923.675} C_VEL
LIN {X 0,Y 592.919,Z 559.862,A -85,B 0,C 180,E1 27920.947,E2 27920.947} C_VEL
LIN {X 0,Y 592.841,Z 579.487,A -85,B 0,C 180,E1 27920.504,E2 27920.504} C_VEL
LIN {X 0,Y 592.742,Z 598.141,A -85,B 0,C 180,E1 27919.896,E2 27919.896} C_VEL
LIN {X 0,Y 592.625,Z 616.45,A -85,B 0,C 180,E1 27919.105,E2 27919.105} C_VEL
LIN {X 0,Y 592.5,Z 634.151,A -85,B 0,C 180,E1 27918.14,E2 27918.14} C_VEL
LIN {X 0,Y 592.37,Z 650.762,A -85,B 0,C 180,E1 27917.025,E2 27917.025} C_VEL
LIN {X 0,Y 592.25,Z 666.231,A -85,B 0,C 180,E1 27915.771,E2 27915.771} C_VEL
LIN {X 0,Y 592.145,Z 680.62,A -85,B 0,C 180,E1 27914.372,E2 27914.372} C_VEL
LIN {X 0,Y 592.064,Z 693.453,A -85,B 0,C 180,E1 27912.88,E2 27912.88} C_VEL
LIN {X 0,Y 592.008,Z 704.786,A -85,B 0,C 180,E1 27911.298,E2 27911.298} C_VEL
LIN {X 0,Y 591.957,Z 714.631,A -85,B 0,C 180,E1 27909.626,E2 27909.626} C_VEL
LIN {X 0,Y 591.933,Z 722.961,A -85,B 0,C 180,E1 27907.864,E2 27907.864} C_VEL
LIN {X 0,Y 591.913,Z 729.701,A -85,B 0,C 180,E1 27906.011,E2 27906.011} C_VEL
LIN {X 0,Y 591.91,Z 734.529,A -85,B 0,C 180,E1 27904.165,E2 27904.165} C_VEL
LIN {X 0,Y 591.914,Z 737.563,A -85,B 0,C 180,E1 27902.323,E2 27902.323} C_VEL
LIN {X 0,Y 591.905,Z 738.907,A -85,B 0,C 180,E1 27900.387,E2 27900.387} C_VEL
LIN {X 0,Y 591.912,Z 738.463,A -85,B 0,C 180,E1 27898.548,E2 27898.548} C_VEL
LIN {X 0,Y 591.915,Z 736.279,A -85,B 0,C 180,E1 27896.676,E2 27896.676} C_VEL
LIN {X 0,Y 591.919,Z 732.451,A -85,B 0,C 180,E1 27894.863,E2 27894.863} C_VEL
LIN {X 0,Y 591.926,Z 726.728,A -85,B 0,C 180,E1 27893.014,E2 27893.014} C_VEL
LIN {X 0,Y 591.947,Z 719.467,A -85,B 0,C 180,E1 27891.256,E2 27891.256} C_VEL
LIN {X 0,Y 591.958,Z 715.339,A -85,B 0,C 180,E1 27890.419,E2 27890.419} C_VEL
LIN {X 0,Y 590.959,Z 711.867,A -85,B 0,C 180,E1 27889.756,E2 27889.756} C_VEL
LIN {X 0,Y 585.038,Z 702.472,A -85,B 0,C 180,E1 27888.117,E2 27888.117} C_VEL
LIN {X 0,Y 584.108,Z 698.186,A -85,B 0,C 180,E1 27887.482,E2 27887.482} C_VEL
LIN {X 0,Y 584.224,Z 685.972,A -85,B 0,C 180,E1 27885.935,E2 27885.935} C_VEL
LIN {X 0,Y 584.365,Z 672.622,A -85,B 0,C 180,E1 27884.519,E2 27884.519} C_VEL
LIN {X 0,Y 584.538,Z 657.783,A -85,B 0,C 180,E1 27883.197,E2 27883.197} C_VEL
LIN {X 0,Y 584.724,Z 641.916,A -85,B 0,C 180,E1 27882.022,E2 27882.022} C_VEL
LIN {X 0,Y 584.918,Z 624.153,A -85,B 0,C 180,E1 27880.943,E2 27880.943} C_VEL
LIN {X 0,Y 585.112,Z 606.068,A -85,B 0,C 180,E1 27880.067,E2 27880.067} C_VEL
LIN {X 0,Y 585.274,Z 587.255,A -85,B 0,C 180,E1 27879.364,E2 27879.364} C_VEL
LIN {X 0,Y 585.408,Z 567.774,A -85,B 0,C 180,E1 27878.839,E2 27878.839} C_VEL
LIN {X 0,Y 585.497,Z 547.656,A -85,B 0,C 180,E1 27878.501,E2 27878.501} C_VEL
LIN {X 0,Y 585.74,Z 344.9,A -85,B 0,C 180,E1 27875.869,E2 27875.869} C_VEL
LIN {X 0,Y 585.285,Z 341.573,A -85,B 0,C 180,E1 27875.764,E2 27875.764} C_VEL
LIN {X 0,Y 585.629,Z 299.36,A -85,B 0,C 180,E1 27872.6,E2 27872.6} C_VEL
LIN {X 0,Y 585.783,Z 269.109,A -85,B 0,C 180,E1 27870.271,E2 27870.271} C_VEL
LIN {X 0,Y 584.062,Z 263.891,A -85,B 0,C 180,E1 27869.724,E2 27869.724} C_VEL
LIN {X 0,Y 584.09,Z 263.714,A -85,B 0,C 180,E1 27866.55,E2 27866.55} C_VEL
LIN {X 0,Y 584.079,Z 263.731,A -85,B 0,C 180,E1 27863.313,E2 27863.313} C_VEL
LIN {X 0,Y 584.064,Z 263.726,A -85,B 0,C 180,E1 27860.061,E2 27860.061} C_VEL
LIN {X 0,Y 584.093,Z 263.727,A -85,B 0,C 180,E1 27856.92,E2 27856.92} C_VEL
LIN {X 0,Y 584.075,Z 263.728,A -85,B 0,C 180,E1 27853.746,E2 27853.746} C_VEL
LIN {X 0,Y 584.097,Z 263.722,A -85,B 0,C 180,E1 27850.45,E2 27850.45} C_VEL
LIN {X 0,Y 584.086,Z 263.729,A -85,B 0,C 180,E1 27847.178,E2 27847.178} C_VEL
LIN {X 0,Y 584.089,Z 263.727,A -85,B 0,C 180,E1 27843.876,E2 27843.876} C_VEL
LIN {X 0,Y 584.077,Z 263.724,A -85,B 0,C 180,E1 27840.674,E2 27840.674} C_VEL
LIN {X 0,Y 584.073,Z 263.73,A -85,B 0,C 180,E1 27837.309,E2 27837.309} C_VEL
LIN {X 0,Y 584.097,Z 263.725,A -85,B 0,C 180,E1 27834.043,E2 27834.043} C_VEL
LIN {X 0,Y 584.051,Z 263.727,A -85,B 0,C 180,E1 27830.861,E2 27830.861} C_VEL
LIN {X 0,Y 584.074,Z 263.732,A -85,B 0,C 180,E1 27827.639,E2 27827.639} C_VEL
LIN {X 0,Y 584.051,Z 263.726,A -85,B 0,C 180,E1 27824.576,E2 27824.576} C_VEL
LIN {X 0,Y 584.033,Z 263.731,A -85,B 0,C 180,E1 27821.355,E2 27821.355} C_VEL
LIN {X 0,Y 584.067,Z 263.734,A -85,B 0,C 180,E1 27818.317,E2 27818.317} C_VEL
LIN {X 0,Y 584.047,Z 263.964,A -85,B 0,C 180,E1 27817.131,E2 27817.131} C_VEL
LIN {X 0,Y 585.523,Z 269.492,A -85,B 0,C 180,E1 27816.62,E2 27816.62} C_VEL
LIN {X 0,Y 585.652,Z 307.821,A -85,B 0,C 180,E1 27813.721,E2 27813.721} C_VEL
LIN {X 0,Y 585.481,Z 340.59,A -85,B 0,C 180,E1 27811.224,E2 27811.224} C_VEL
LIN {X 0,Y 585.116,Z 381.223,A -85,B 0,C 180,E1 27808.141,E2 27808.141} C_VEL
LIN {X 0,Y 584.848,Z 422.816,A -85,B 0,C 180,E1 27805.048,E2 27805.048} C_VEL
LIN {X 0,Y 584.548,Z 467.504,A -85,B 0,C 180,E1 27801.79,E2 27801.79} C_VEL
LIN {X 0,Y 584.606,Z 472.889,A -85,B 0,C 180,E1 27801.438,E2 27801.438} C_VEL
LIN {X 0,Y 584.78,Z 515.756,A -85,B 0,C 180,E1 27800.891,E2 27800.891} C_VEL
LIN {X 0,Y 584.627,Z 615.439,A -85,B 0,C 180,E1 27799.625,E2 27799.625} C_VEL
LIN {X 0,Y 584.579,Z 632.194,A -85,B 0,C 180,E1 27799.216,E2 27799.216} C_VEL
LIN {X 0,Y 584.479,Z 647.54,A -85,B 0,C 180,E1 27798.656,E2 27798.656} C_VEL
LIN {X 0,Y 584.367,Z 662.663,A -85,B 0,C 180,E1 27797.902,E2 27797.902} C_VEL
LIN {X 0,Y 584.266,Z 676.67,A -85,B 0,C 180,E1 27797.004,E2 27797.004} C_VEL
LIN {X 0,Y 584.154,Z 689.816,A -85,B 0,C 180,E1 27795.935,E2 27795.935} C_VEL
LIN {X 0,Y 584.07,Z 701.828,A -85,B 0,C 180,E1 27794.716,E2 27794.716} C_VEL
LIN {X 0,Y 584.002,Z 712.233,A -85,B 0,C 180,E1 27793.388,E2 27793.388} C_VEL
LIN {X 0,Y 583.96,Z 721.139,A -85,B 0,C 180,E1 27791.948,E2 27791.948} C_VEL
LIN {X 0,Y 583.93,Z 728.436,A -85,B 0,C 180,E1 27790.392,E2 27790.392} C_VEL
LIN {X 0,Y 583.919,Z 733.459,A -85,B 0,C 180,E1 27788.927,E2 27788.927} C_VEL
LIN {X 0,Y 583.914,Z 736.995,A -85,B 0,C 180,E1 27787.341,E2 27787.341} C_VEL
LIN {X 0,Y 583.917,Z 738.77,A -85,B 0,C 180,E1 27785.736,E2 27785.736} C_VEL
LIN {X 0,Y 583.915,Z 738.802,A -85,B 0,C 180,E1 27784.22,E2 27784.22} C_VEL
LIN {X 0,Y 583.915,Z 737.002,A -85,B 0,C 180,E1 27782.575,E2 27782.575} C_VEL
LIN {X 0,Y 583.919,Z 733.555,A -85,B 0,C 180,E1 27781.016,E2 27781.016} C_VEL
LIN {X 0,Y 583.932,Z 728.092,A -85,B 0,C 180,E1 27779.434,E2 27779.434} C_VEL
LIN {X 0,Y 583.959,Z 721.04,A -85,B 0,C 180,E1 27777.943,E2 27777.943} C_VEL
LIN {X 0,Y 584.001,Z 712.401,A -85,B 0,C 180,E1 27776.546,E2 27776.546} C_VEL
LIN {X 0,Y 584.072,Z 701.775,A -85,B 0,C 180,E1 27775.188,E2 27775.188} C_VEL
LIN {X 0,Y 584.153,Z 689.981,A -85,B 0,C 180,E1 27773.99,E2 27773.99} C_VEL
LIN {X 0,Y 584.257,Z 677.416,A -85,B 0,C 180,E1 27772.961,E2 27772.961} C_VEL
LIN {X 0,Y 584.36,Z 663.378,A -85,B 0,C 180,E1 27772.048,E2 27772.048} C_VEL
LIN {X 0,Y 584.47,Z 647.873,A -85,B 0,C 180,E1 27771.269,E2 27771.269} C_VEL
LIN {X 0,Y 584.578,Z 631.879,A -85,B 0,C 180,E1 27770.684,E2 27770.684} C_VEL
LIN {X 0,Y 584.615,Z 614.997,A -85,B 0,C 180,E1 27770.276,E2 27770.276} C_VEL
LIN {X 0,Y 584.627,Z 473.187,A -85,B 0,C 180,E1 27768.479,E2 27768.479} C_VEL
LIN {X 0,Y 584.513,Z 470.309,A -85,B 0,C 180,E1 27768.322,E2 27768.322} C_VEL
LIN {X 0,Y 584.768,Z 429.353,A -85,B 0,C 180,E1 27765.341,E2 27765.341} C_VEL
LIN {X 0,Y 585.047,Z 385.978,A -85,B 0,C 180,E1 27762.125,E2 27762.125} C_VEL
LIN {X 0,Y 585.448,Z 346.351,A -85,B 0,C 180,E1 27759.128,E2 27759.128} C_VEL
LIN {X 0,Y 585.638,Z 312.865,A -85,B 0,C 180,E1 27756.574,E2 27756.574} C_VEL
LIN {X 0,Y 585.451,Z 273.865,A -85,B 0,C 180,E1 27753.656,E2 27753.656} C_VEL
LIN {X 0,Y 585.195,Z 267.775,A -85,B 0,C 180,E1 27753.203,E2 27753.203} C_VEL
LIN {X 0,Y 584.083,Z 263.947,A -85,B 0,C 180,E1 27752.835,E2 27752.835} C_VEL
LIN {X 0,Y 584.101,Z 263.731,A -85,B 0,C 180,E1 27749.764,E2 27749.764} C_VEL
LIN {X 0,Y 584.049,Z 263.729,A -85,B 0,C 180,E1 27746.54,E2 27746.54} C_VEL
LIN {X 0,Y 584.097,Z 263.726,A -85,B 0,C 180,E1 27743.293,E2 27743.293} C_VEL
LIN {X 0,Y 584.061,Z 263.729,A -85,B 0,C 180,E1 27740.127,E2 27740.127} C_VEL
LIN {X 0,Y 584.062,Z 263.726,A -85,B 0,C 180,E1 27736.817,E2 27736.817} C_VEL
LIN {X 0,Y 584.094,Z 263.733,A -85,B 0,C 180,E1 27733.665,E2 27733.665} C_VEL
LIN {X 0,Y 584.052,Z 263.727,A -85,B 0,C 180,E1 27730.456,E2 27730.456} C_VEL
LIN {X 0,Y 584.098,Z 263.726,A -85,B 0,C 180,E1 27727.278,E2 27727.278} C_VEL
LIN {X 0,Y 584.056,Z 263.729,A -85,B 0,C 180,E1 27724.124,E2 27724.124} C_VEL
LIN {X 0,Y 584.086,Z 263.724,A -85,B 0,C 180,E1 27720.883,E2 27720.883} C_VEL
LIN {X 0,Y 584.085,Z 263.731,A -85,B 0,C 180,E1 27717.646,E2 27717.646} C_VEL
LIN {X 0,Y 584.058,Z 263.726,A -85,B 0,C 180,E1 27714.401,E2 27714.401} C_VEL
LIN {X 0,Y 584.097,Z 263.727,A -85,B 0,C 180,E1 27711.237,E2 27711.237} C_VEL
LIN {X 0,Y 584.057,Z 263.728,A -85,B 0,C 180,E1 27708.045,E2 27708.045} C_VEL
LIN {X 0,Y 584.095,Z 263.723,A -85,B 0,C 180,E1 27704.817,E2 27704.817} C_VEL
LIN {X 0,Y 584.089,Z 263.731,A -85,B 0,C 180,E1 27701.499,E2 27701.499} C_VEL
LIN {X 0,Y 584.059,Z 263.726,A -85,B 0,C 180,E1 27698.193,E2 27698.193} C_VEL
LIN {X 0,Y 584.096,Z 263.726,A -85,B 0,C 180,E1 27694.988,E2 27694.988} C_VEL
LIN {X 0,Y 584.062,Z 263.728,A -85,B 0,C 180,E1 27691.805,E2 27691.805} C_VEL
LIN {X 0,Y 584.084,Z 263.723,A -85,B 0,C 180,E1 27688.481,E2 27688.481} C_VEL
LIN {X 0,Y 584.092,Z 263.732,A -85,B 0,C 180,E1 27685.248,E2 27685.248} C_VEL
LIN {X 0,Y 584.063,Z 263.726,A -85,B 0,C 180,E1 27682.079,E2 27682.079} C_VEL
LIN {X 0,Y 584.095,Z 263.728,A -85,B 0,C 180,E1 27678.903,E2 27678.903} C_VEL
LIN {X 0,Y 584.064,Z 263.729,A -85,B 0,C 180,E1 27675.688,E2 27675.688} C_VEL
LIN {X 0,Y 584.092,Z 263.724,A -85,B 0,C 180,E1 27672.41,E2 27672.41} C_VEL
LIN {X 0,Y 584.101,Z 263.731,A -85,B 0,C 180,E1 27669.044,E2 27669.044} C_VEL
LIN {X 0,Y 584.062,Z 263.717,A -85,B 0,C 180,E1 27665.834,E2 27665.834} C_VEL
LIN {X 0,Y 584.093,Z 263.712,A -85,B 0,C 180,E1 27662.626,E2 27662.626} C_VEL
LIN {X 0,Y 584.183,Z 264.259,A -85,B 0,C 180,E1 27662.367,E2 27662.367} C_VEL
LIN {X 0,Y 586.429,Z 270.435,A -85,B 0,C 180,E1 27661.791,E2 27661.791} C_VEL
LIN {X 0,Y 586.03,Z 315.223,A -85,B 0,C 180,E1 27658.824,E2 27658.824} C_VEL
LIN {X 0,Y 586.68,Z 320.862,A -85,B 0,C 180,E1 27658.702,E2 27658.702} C_VEL
LIN {X 0,Y 586.149,Z 549.886,A -85,B 0,C 180,E1 27655.64,E2 27655.64} C_VEL
LIN {X 0,Y 586.038,Z 580.239,A -85,B 0,C 180,E1 27655.196,E2 27655.196} C_VEL
LIN {X 0,Y 585.897,Z 600.76,A -85,B 0,C 180,E1 27654.713,E2 27654.713} C_VEL
LIN {X 0,Y 585.704,Z 621.201,A -85,B 0,C 180,E1 27654.035,E2 27654.035} C_VEL
LIN {X 0,Y 585.478,Z 639.884,A -85,B 0,C 180,E1 27653.233,E2 27653.233} C_VEL
LIN {X 0,Y 585.23,Z 658.759,A -85,B 0,C 180,E1 27652.235,E2 27652.235} C_VEL
LIN {X 0,Y 584.98,Z 677.48,A -85,B 0,C 180,E1 27651.033,E2 27651.033} C_VEL
LIN {X 0,Y 584.755,Z 694.592,A -85,B 0,C 180,E1 27649.721,E2 27649.721} C_VEL
LIN {X 0,Y 584.555,Z 710.114,A -85,B 0,C 180,E1 27648.322,E2 27648.322} C_VEL
LIN {X 0,Y 584.368,Z 725.364,A -85,B 0,C 180,E1 27646.704,E2 27646.704} C_VEL
LIN {X 0,Y 584.207,Z 739.14,A -85,B 0,C 180,E1 27644.976,E2 27644.976} C_VEL
LIN {X 0,Y 584.09,Z 751.3,A -85,B 0,C 180,E1 27643.159,E2 27643.159} C_VEL
LIN {X 0,Y 584.011,Z 761.37,A -85,B 0,C 180,E1 27641.354,E2 27641.354} C_VEL
LIN {X 0,Y 583.957,Z 770.066,A -85,B 0,C 180,E1 27639.46,E2 27639.46} C_VEL
LIN {X 0,Y 583.926,Z 777.192,A -85,B 0,C 180,E1 27637.511,E2 27637.511} C_VEL
LIN {X 0,Y 583.914,Z 782.51,A -85,B 0,C 180,E1 27635.6,E2 27635.6} C_VEL
LIN {X 0,Y 583.907,Z 786.243,A -85,B 0,C 180,E1 27633.631,E2 27633.631} C_VEL
LIN {X 0,Y 583.904,Z 788.374,A -85,B 0,C 180,E1 27631.667,E2 27631.667} C_VEL
LIN {X 0,Y 583.9,Z 788.917,A -85,B 0,C 180,E1 27629.606,E2 27629.606} C_VEL
LIN {X 0,Y 583.905,Z 787.838,A -85,B 0,C 180,E1 27627.644,E2 27627.644} C_VEL
LIN {X 0,Y 583.908,Z 784.971,A -85,B 0,C 180,E1 27625.58,E2 27625.58} C_VEL
LIN {X 0,Y 583.92,Z 780.48,A -85,B 0,C 180,E1 27623.609,E2 27623.609} C_VEL
LIN {X 0,Y 583.943,Z 774.262,A -85,B 0,C 180,E1 27621.63,E2 27621.63} C_VEL
LIN {X 0,Y 583.984,Z 766.173,A -85,B 0,C 180,E1 27619.642,E2 27619.642} C_VEL
LIN {X 0,Y 584.049,Z 756.563,A -85,B 0,C 180,E1 27617.743,E2 27617.743} C_VEL
LIN {X 0,Y 584.148,Z 745.491,A -85,B 0,C 180,E1 27615.932,E2 27615.932} C_VEL
LIN {X 0,Y 584.272,Z 732.93,A -85,B 0,C 180,E1 27614.21,E2 27614.21} C_VEL
LIN {X 0,Y 584.436,Z 718.879,A -85,B 0,C 180,E1 27612.578,E2 27612.578} C_VEL
LIN {X 0,Y 584.624,Z 703.836,A -85,B 0,C 180,E1 27611.088,E2 27611.088} C_VEL
LIN {X 0,Y 584.844,Z 687.279,A -85,B 0,C 180,E1 27609.692,E2 27609.692} C_VEL
LIN {X 0,Y 585.085,Z 669.738,A -85,B 0,C 180,E1 27608.443,E2 27608.443} C_VEL
LIN {X 0,Y 585.339,Z 651.251,A -85,B 0,C 180,E1 27607.343,E2 27607.343} C_VEL
LIN {X 0,Y 585.578,Z 633.055,A -85,B 0,C 180,E1 27606.449,E2 27606.449} C_VEL
LIN {X 0,Y 585.764,Z 613.629,A -85,B 0,C 180,E1 27605.692,E2 27605.692} C_VEL
LIN {X 0,Y 585.938,Z 593.746,A -85,B 0,C 180,E1 27605.104,E2 27605.104} C_VEL
LIN {X 0,Y 586.085,Z 572.695,A -85,B 0,C 180,E1 27604.675,E2 27604.675} C_VEL
LIN {X 0,Y 586.658,Z 330.991,A -85,B 0,C 180,E1 27601.435,E2 27601.435} C_VEL
LIN {X 0,Y 586.455,Z 317.862,A -85,B 0,C 180,E1 27601.245,E2 27601.245} C_VEL
LIN {X 0,Y 586.013,Z 314.36,A -85,B 0,C 180,E1 27601.127,E2 27601.127} C_VEL
LIN {X 0,Y 586.423,Z 270.398,A -85,B 0,C 180,E1 27598.206,E2 27598.206} C_VEL
LIN {X 0,Y 584.143,Z 264.042,A -85,B 0,C 180,E1 27597.604,E2 27597.604} C_VEL
LIN {X 0,Y 584.087,Z 263.723,A -85,B 0,C 180,E1 27596.833,E2 27596.833} C_VEL
LIN {X 0,Y 584.097,Z 263.726,A -85,B 0,C 180,E1 27593.558,E2 27593.558} C_VEL
LIN {X 0,Y 584.058,Z 263.729,A -85,B 0,C 180,E1 27590.316,E2 27590.316} C_VEL
LIN {X 0,Y 584.097,Z 263.731,A -85,B 0,C 180,E1 27587.109,E2 27587.109} C_VEL
LIN {X 0,Y 584.057,Z 263.728,A -85,B 0,C 180,E1 27584.027,E2 27584.027} C_VEL
LIN {X 0,Y 584.074,Z 263.732,A -85,B 0,C 180,E1 27580.709,E2 27580.709} C_VEL
LIN {X 0,Y 584.086,Z 263.726,A -85,B 0,C 180,E1 27577.547,E2 27577.547} C_VEL
LIN {X 0,Y 584.051,Z 263.732,A -85,B 0,C 180,E1 27574.395,E2 27574.395} C_VEL
LIN {X 0,Y 584.099,Z 263.724,A -85,B 0,C 180,E1 27571.243,E2 27571.243} C_VEL
LIN {X 0,Y 584.072,Z 263.937,A -85,B 0,C 180,E1 27570.174,E2 27570.174} C_VEL
LIN {X 0,Y 585.933,Z 270.168,A -85,B 0,C 180,E1 27569.548,E2 27569.548} C_VEL
LIN {X 0,Y 585.51,Z 310.492,A -85,B 0,C 180,E1 27566.468,E2 27566.468} C_VEL
LIN {X 0,Y 585.352,Z 342.589,A -85,B 0,C 180,E1 27564.094,E2 27564.094} C_VEL
LIN {X 0,Y 585.885,Z 347.766,A -85,B 0,C 180,E1 27563.997,E2 27563.997} C_VEL
LIN {X 0,Y 585.445,Z 559.888,A -85,B 0,C 180,E1 27561.227,E2 27561.227} C_VEL
LIN {X 0,Y 585.327,Z 579.62,A -85,B 0,C 180,E1 27560.776,E2 27560.776} C_VEL
LIN {X 0,Y 585.167,Z 598.8,A -85,B 0,C 180,E1 27560.139,E2 27560.139} C_VEL
LIN {X 0,Y 584.985,Z 617.38,A -85,B 0,C 180,E1 27559.318,E2 27559.318} C_VEL
LIN {X 0,Y 584.796,Z 634.971,A -85,B 0,C 180,E1 27558.336,E2 27558.336} C_VEL
LIN {X 0,Y 584.604,Z 651.393,A -85,B 0,C 180,E1 27557.21,E2 27557.21} C_VEL
LIN {X 0,Y 584.428,Z 666.638,A -85,B 0,C 180,E1 27555.952,E2 27555.952} C_VEL
LIN {X 0,Y 584.27,Z 680.625,A -85,B 0,C 180,E1 27554.57,E2 27554.57} C_VEL
LIN {X 0,Y 584.146,Z 693.461,A -85,B 0,C 180,E1 27553.058,E2 27553.058} C_VEL
LIN {X 0,Y 584.056,Z 704.794,A -85,B 0,C 180,E1 27551.454,E2 27551.454} C_VEL
LIN {X 0,Y 583.982,Z 714.637,A -85,B 0,C 180,E1 27549.759,E2 27549.759} C_VEL
LIN {X 0,Y 583.946,Z 722.963,A -85,B 0,C 180,E1 27547.972,E2 27547.972} C_VEL
LIN {X 0,Y 583.919,Z 729.705,A -85,B 0,C 180,E1 27546.094,E2 27546.094} C_VEL
LIN {X 0,Y 583.909,Z 734.533,A -85,B 0,C 180,E1 27544.222,E2 27544.222} C_VEL
LIN {X 0,Y 583.914,Z 737.566,A -85,B 0,C 180,E1 27542.355,E2 27542.355} C_VEL
LIN {X 0,Y 583.905,Z 738.907,A -85,B 0,C 180,E1 27540.392,E2 27540.392} C_VEL
LIN {X 0,Y 583.912,Z 738.464,A -85,B 0,C 180,E1 27538.528,E2 27538.528} C_VEL
LIN {X 0,Y 583.915,Z 736.322,A -85,B 0,C 180,E1 27536.656,E2 27536.656} C_VEL
LIN {X 0,Y 583.92,Z 732.452,A -85,B 0,C 180,E1 27534.793,E2 27534.793} C_VEL
LIN {X 0,Y 583.936,Z 726.727,A -85,B 0,C 180,E1 27532.918,E2 27532.918} C_VEL
LIN {X 0,Y 583.966,Z 719.004,A -85,B 0,C 180,E1 27531.036,E2 27531.036} C_VEL
LIN {X 0,Y 584.018,Z 709.624,A -85,B 0,C 180,E1 27529.244,E2 27529.244} C_VEL
LIN {X 0,Y 584.095,Z 699.324,A -85,B 0,C 180,E1 27527.644,E2 27527.644} C_VEL
LIN {X 0,Y 584.108,Z 698.186,A -85,B 0,C 180,E1 27527.482,E2 27527.482} C_VEL
LIN {X 0,Y 583.191,Z 693.811,A -85,B 0,C 180,E1 27526.859,E2 27526.859} C_VEL
LIN {X 0,Y 577.405,Z 682.292,A -85,B 0,C 180,E1 27525.329,E2 27525.329} C_VEL
LIN {X 0,Y 576.462,Z 677.121,A -85,B 0,C 180,E1 27524.76,E2 27524.76} C_VEL
LIN {X 0,Y 576.677,Z 662.603,A -85,B 0,C 180,E1 27523.376,E2 27523.376} C_VEL
LIN {X 0,Y 576.922,Z 647.026,A -85,B 0,C 180,E1 27522.136,E2 27522.136} C_VEL
LIN {X 0,Y 577.169,Z 630.739,A -85,B 0,C 180,E1 27521.062,E2 27521.062} C_VEL
LIN {X 0,Y 577.424,Z 613.289,A -85,B 0,C 180,E1 27520.126,E2 27520.126} C_VEL
LIN {X 0,Y 577.656,Z 595.368,A -85,B 0,C 180,E1 27519.366,E2 27519.366} C_VEL
LIN {X 0,Y 577.86,Z 576.166,A -85,B 0,C 180,E1 27518.758,E2 27518.758} C_VEL
LIN {X 0,Y 578.008,Z 557.027,A -85,B 0,C 180,E1 27518.348,E2 27518.348} C_VEL
LIN {X 0,Y 578.445,Z 346.121,A -85,B 0,C 180,E1 27515.562,E2 27515.562} C_VEL
LIN {X 0,Y 577.781,Z 342.045,A -85,B 0,C 180,E1 27515.46,E2 27515.46} C_VEL
LIN {X 0,Y 578.245,Z 300.128,A -85,B 0,C 180,E1 27512.281,E2 27512.281} C_VEL
LIN {X 0,Y 578.472,Z 272.066,A -85,B 0,C 180,E1 27510.092,E2 27510.092} C_VEL
LIN {X 0,Y 576.148,Z 264.916,A -85,B 0,C 180,E1 27509.353,E2 27509.353} C_VEL
LIN {X 0,Y 576.111,Z 264.701,A -85,B 0,C 180,E1 27506.024,E2 27506.024} C_VEL
LIN {X 0,Y 576.16,Z 264.716,A -85,B 0,C 180,E1 27502.849,E2 27502.849} C_VEL
LIN {X 0,Y 576.128,Z 264.718,A -85,B 0,C 180,E1 27499.631,E2 27499.631} C_VEL
LIN {X 0,Y 576.145,Z 264.713,A -85,B 0,C 180,E1 27496.314,E2 27496.314} C_VEL
LIN {X 0,Y 576.15,Z 264.717,A -85,B 0,C 180,E1 27493.002,E2 27493.002} C_VEL
LIN {X 0,Y 576.144,Z 264.717,A -85,B 0,C 180,E1 27489.753,E2 27489.753} C_VEL
LIN {X 0,Y 576.158,Z 264.711,A -85,B 0,C 180,E1 27486.407,E2 27486.407} C_VEL
LIN {X 0,Y 576.138,Z 264.717,A -85,B 0,C 180,E1 27483.139,E2 27483.139} C_VEL
LIN {X 0,Y 576.155,Z 264.716,A -85,B 0,C 180,E1 27479.873,E2 27479.873} C_VEL
LIN {X 0,Y 576.134,Z 264.714,A -85,B 0,C 180,E1 27476.6,E2 27476.6} C_VEL
LIN {X 0,Y 576.125,Z 264.719,A -85,B 0,C 180,E1 27473.31,E2 27473.31} C_VEL
LIN {X 0,Y 576.161,Z 264.715,A -85,B 0,C 180,E1 27470.098,E2 27470.098} C_VEL
LIN {X 0,Y 576.102,Z 264.719,A -85,B 0,C 180,E1 27466.953,E2 27466.953} C_VEL
LIN {X 0,Y 576.136,Z 264.713,A -85,B 0,C 180,E1 27463.755,E2 27463.755} C_VEL
LIN {X 0,Y 576.096,Z 264.719,A -85,B 0,C 180,E1 27460.703,E2 27460.703} C_VEL
LIN {X 0,Y 576.102,Z 264.798,A -85,B 0,C 180,E1 27457.48,E2 27457.48} C_VEL
LIN {X 0,Y 576.549,Z 266.601,A -85,B 0,C 180,E1 27457.262,E2 27457.262} C_VEL
LIN {X 0,Y 578.054,Z 272.367,A -85,B 0,C 180,E1 27456.756,E2 27456.756} C_VEL
LIN {X 0,Y 578.093,Z 311.497,A -85,B 0,C 180,E1 27453.769,E2 27453.769} C_VEL
LIN {X 0,Y 577.913,Z 352.736,A -85,B 0,C 180,E1 27450.645,E2 27450.645} C_VEL
LIN {X 0,Y 577.434,Z 393.635,A -85,B 0,C 180,E1 27447.52,E2 27447.52} C_VEL
LIN {X 0,Y 577.022,Z 438.206,A -85,B 0,C 180,E1 27444.183,E2 27444.183} C_VEL
LIN {X 0,Y 576.787,Z 472.434,A -85,B 0,C 180,E1 27441.679,E2 27441.679} C_VEL
LIN {X 0,Y 577.159,Z 479.84,A -85,B 0,C 180,E1 27441.564,E2 27441.564} C_VEL
LIN {X 0,Y 576.884,Z 615.467,A -85,B 0,C 180,E1 27439.826,E2 27439.826} C_VEL
LIN {X 0,Y 576.81,Z 632.149,A -85,B 0,C 180,E1 27439.413,E2 27439.413} C_VEL
LIN {X 0,Y 576.685,Z 647.298,A -85,B 0,C 180,E1 27438.855,E2 27438.855} C_VEL
LIN {X 0,Y 576.528,Z 662.503,A -85,B 0,C 180,E1 27438.091,E2 27438.091} C_VEL
LIN {X 0,Y 576.388,Z 676.649,A -85,B 0,C 180,E1 27437.172,E2 27437.172} C_VEL
LIN {X 0,Y 576.244,Z 689.721,A -85,B 0,C 180,E1 27436.096,E2 27436.096} C_VEL
LIN {X 0,Y 576.131,Z 701.3,A -85,B 0,C 180,E1 27434.912,E2 27434.912} C_VEL
LIN {X 0,Y 576.037,Z 711.807,A -85,B 0,C 180,E1 27433.566,E2 27433.566} C_VEL
LIN {X 0,Y 575.977,Z 720.813,A -85,B 0,C 180,E1 27432.107,E2 27432.107} C_VEL
LIN {X 0,Y 575.939,Z 727.754,A -85,B 0,C 180,E1 27430.636,E2 27430.636} C_VEL
LIN {X 0,Y 575.923,Z 733.265,A -85,B 0,C 180,E1 27429.046,E2 27429.046} C_VEL
LIN {X 0,Y 575.917,Z 736.857,A -85,B 0,C 180,E1 27427.462,E2 27427.462} C_VEL
LIN {X 0,Y 575.918,Z 738.726,A -85,B 0,C 180,E1 27425.814,E2 27425.814} C_VEL
LIN {X 0,Y 575.915,Z 738.844,A -85,B 0,C 180,E1 27424.278,E2 27424.278} C_VEL
LIN {X 0,Y 575.915,Z 737.109,A -85,B 0,C 180,E1 27422.61,E2 27422.61} C_VEL
LIN {X 0,Y 575.92,Z 733.738,A -85,B 0,C 180,E1 27421.03,E2 27421.03} C_VEL
LIN {X 0,Y 575.938,Z 728.373,A -85,B 0,C 180,E1 27419.427,E2 27419.427} C_VEL
LIN {X 0,Y 575.973,Z 721.338,A -85,B 0,C 180,E1 27417.903,E2 27417.903} C_VEL
LIN {X 0,Y 576.029,Z 712.879,A -85,B 0,C 180,E1 27416.499,E2 27416.499} C_VEL
LIN {X 0,Y 576.121,Z 702.422,A -85,B 0,C 180,E1 27415.129,E2 27415.129} C_VEL
LIN {X 0,Y 576.233,Z 690.822,A -85,B 0,C 180,E1 27413.916,E2 27413.916} C_VEL
LIN {X 0,Y 576.376,Z 677.75,A -85,B 0,C 180,E1 27412.82,E2 27412.82} C_VEL
LIN {X 0,Y 576.508,Z 664.634,A -85,B 0,C 180,E1 27411.943,E2 27411.943} C_VEL
LIN {X 0,Y 576.648,Z 649.686,A -85,B 0,C 180,E1 27411.162,E2 27411.162} C_VEL
LIN {X 0,Y 576.795,Z 633.926,A -85,B 0,C 180,E1 27410.553,E2 27410.553} C_VEL
LIN {X 0,Y 576.868,Z 617.413,A -85,B 0,C 180,E1 27410.122,E2 27410.122} C_VEL
LIN {X 0,Y 576.913,Z 591.139,A -85,B 0,C 180,E1 27409.75,E2 27409.75} C_VEL
LIN {X 0,Y 576.946,Z 473.984,A -85,B 0,C 180,E1 27408.265,E2 27408.265} C_VEL
LIN {X 0,Y 576.748,Z 471.856,A -85,B 0,C 180,E1 27408.199,E2 27408.199} C_VEL
LIN {X 0,Y 577.064,Z 431.503,A -85,B 0,C 180,E1 27405.229,E2 27405.229} C_VEL
LIN {X 0,Y 577.457,Z 388.314,A -85,B 0,C 180,E1 27401.986,E2 27401.986} C_VEL
LIN {X 0,Y 577.962,Z 348.869,A -85,B 0,C 180,E1 27398.966,E2 27398.966} C_VEL
LIN {X 0,Y 578.032,Z 306.453,A -85,B 0,C 180,E1 27395.78,E2 27395.78} C_VEL
LIN {X 0,Y 577.91,Z 276.15,A -85,B 0,C 180,E1 27393.499,E2 27393.499} C_VEL
LIN {X 0,Y 577.638,Z 270.109,A -85,B 0,C 180,E1 27393.042,E2 27393.042} C_VEL
LIN {X 0,Y 576.147,Z 264.988,A -85,B 0,C 180,E1 27392.562,E2 27392.562} C_VEL
LIN {X 0,Y 576.136,Z 264.722,A -85,B 0,C 180,E1 27389.988,E2 27389.988} C_VEL
LIN {X 0,Y 576.113,Z 264.717,A -85,B 0,C 180,E1 27386.712,E2 27386.712} C_VEL
LIN {X 0,Y 576.161,Z 264.718,A -85,B 0,C 180,E1 27383.525,E2 27383.525} C_VEL
LIN {X 0,Y 576.113,Z 264.717,A -85,B 0,C 180,E1 27380.311,E2 27380.311} C_VEL
LIN {X 0,Y 576.14,Z 264.715,A -85,B 0,C 180,E1 27377.021,E2 27377.021} C_VEL
LIN {X 0,Y 576.139,Z 264.72,A -85,B 0,C 180,E1 27373.857,E2 27373.857} C_VEL
LIN {X 0,Y 576.117,Z 264.715,A -85,B 0,C 180,E1 27370.601,E2 27370.601} C_VEL
LIN {X 0,Y 576.16,Z 264.717,A -85,B 0,C 180,E1 27367.379,E2 27367.379} C_VEL
LIN {X 0,Y 576.116,Z 264.717,A -85,B 0,C 180,E1 27364.18,E2 27364.18} C_VEL
LIN {X 0,Y 576.148,Z 264.713,A -85,B 0,C 180,E1 27360.895,E2 27360.895} C_VEL
LIN {X 0,Y 576.149,Z 264.72,A -85,B 0,C 180,E1 27357.613,E2 27357.613} C_VEL
LIN {X 0,Y 576.117,Z 264.716,A -85,B 0,C 180,E1 27354.323,E2 27354.323} C_VEL
LIN {X 0,Y 576.159,Z 264.714,A -85,B 0,C 180,E1 27351.115,E2 27351.115} C_VEL
LIN {X 0,Y 576.124,Z 264.718,A -85,B 0,C 180,E1 27347.878,E2 27347.878} C_VEL
LIN {X 0,Y 576.131,Z 264.713,A -85,B 0,C 180,E1 27344.499,E2 27344.499} C_VEL
LIN {X 0,Y 576.159,Z 264.719,A -85,B 0,C 180,E1 27341.274,E2 27341.274} C_VEL
LIN {X 0,Y 576.119,Z 264.715,A -85,B 0,C 180,E1 27338.091,E2 27338.091} C_VEL
LIN {X 0,Y 576.158,Z 264.713,A -85,B 0,C 180,E1 27334.839,E2 27334.839} C_VEL
LIN {X 0,Y 576.133,Z 264.718,A -85,B 0,C 180,E1 27331.607,E2 27331.607} C_VEL
LIN {X 0,Y 576.129,Z 264.714,A -85,B 0,C 180,E1 27328.25,E2 27328.25} C_VEL
LIN {X 0,Y 576.157,Z 264.717,A -85,B 0,C 180,E1 27324.992,E2 27324.992} C_VEL
LIN {X 0,Y 576.122,Z 264.716,A -85,B 0,C 180,E1 27321.827,E2 27321.827} C_VEL
LIN {X 0,Y 576.159,Z 264.712,A -85,B 0,C 180,E1 27318.561,E2 27318.561} C_VEL
LIN {X 0,Y 576.155,Z 264.72,A -85,B 0,C 180,E1 27315.205,E2 27315.205} C_VEL
LIN {X 0,Y 576.125,Z 264.717,A -85,B 0,C 180,E1 27311.882,E2 27311.882} C_VEL
LIN {X 0,Y 576.156,Z 264.716,A -85,B 0,C 180,E1 27308.655,E2 27308.655} C_VEL
LIN {X 0,Y 576.131,Z 264.701,A -85,B 0,C 180,E1 27305.424,E2 27305.424} C_VEL
LIN {X 0,Y 576.191,Z 264.963,A -85,B 0,C 180,E1 27302.847,E2 27302.847} C_VEL
LIN {X 0,Y 579.319,Z 273.816,A -85,B 0,C 180,E1 27301.994,E2 27301.994} C_VEL
LIN {X 0,Y 578.843,Z 315.684,A -85,B 0,C 180,E1 27299.204,E2 27299.204} C_VEL
LIN {X 0,Y 579.658,Z 322.135,A -85,B 0,C 180,E1 27299.065,E2 27299.065} C_VEL
LIN {X 0,Y 578.931,Z 551.159,A -85,B 0,C 180,E1 27295.966,E2 27295.966} C_VEL
LIN {X 0,Y 578.782,Z 580.563,A -85,B 0,C 180,E1 27295.527,E2 27295.527} C_VEL
LIN {X 0,Y 578.596,Z 600.975,A -85,B 0,C 180,E1 27295.04,E2 27295.04} C_VEL
LIN {X 0,Y 578.344,Z 620.736,A -85,B 0,C 180,E1 27294.378,E2 27294.378} C_VEL
LIN {X 0,Y 578.032,Z 640.069,A -85,B 0,C 180,E1 27293.541,E2 27293.541} C_VEL
LIN {X 0,Y 577.706,Z 658.883,A -85,B 0,C 180,E1 27292.533,E2 27292.533} C_VEL
LIN {X 0,Y 577.367,Z 677.791,A -85,B 0,C 180,E1 27291.302,E2 27291.302} C_VEL
LIN {X 0,Y 577.055,Z 695.027,A -85,B 0,C 180,E1 27289.957,E2 27289.957} C_VEL
LIN {X 0,Y 576.768,Z 710.925,A -85,B 0,C 180,E1 27288.495,E2 27288.495} C_VEL
LIN {X 0,Y 576.53,Z 725.365,A -85,B 0,C 180,E1 27286.938,E2 27286.938} C_VEL
LIN {X 0,Y 576.317,Z 739.139,A -85,B 0,C 180,E1 27285.186,E2 27285.186} C_VEL
LIN {X 0,Y 576.152,Z 751.299,A -85,B 0,C 180,E1 27283.343,E2 27283.343} C_VEL
LIN {X 0,Y 576.044,Z 761.371,A -85,B 0,C 180,E1 27281.513,E2 27281.513} C_VEL
LIN {X 0,Y 575.975,Z 770.066,A -85,B 0,C 180,E1 27279.592,E2 27279.592} C_VEL
LIN {X 0,Y 575.943,Z 776.994,A -85,B 0,C 180,E1 27277.681,E2 27277.681} C_VEL
LIN {X 0,Y 575.92,Z 782.511,A -85,B 0,C 180,E1 27275.678,E2 27275.678} C_VEL
LIN {X 0,Y 575.91,Z 786.243,A -85,B 0,C 180,E1 27273.682,E2 27273.682} C_VEL
LIN {X 0,Y 575.905,Z 788.374,A -85,B 0,C 180,E1 27271.69,E2 27271.69} C_VEL
LIN {X 0,Y 575.9,Z 788.917,A -85,B 0,C 180,E1 27269.601,E2 27269.601} C_VEL
LIN {X 0,Y 575.905,Z 787.838,A -85,B 0,C 180,E1 27267.611,E2 27267.611} C_VEL
LIN {X 0,Y 575.911,Z 784.971,A -85,B 0,C 180,E1 27265.518,E2 27265.518} C_VEL
LIN {X 0,Y 575.924,Z 780.481,A -85,B 0,C 180,E1 27263.52,E2 27263.52} C_VEL
LIN {X 0,Y 575.954,Z 774.262,A -85,B 0,C 180,E1 27261.513,E2 27261.513} C_VEL
LIN {X 0,Y 576.006,Z 766.174,A -85,B 0,C 180,E1 27259.497,E2 27259.497} C_VEL
LIN {X 0,Y 576.095,Z 756.562,A -85,B 0,C 180,E1 27257.571,E2 27257.571} C_VEL
LIN {X 0,Y 576.234,Z 745.489,A -85,B 0,C 180,E1 27255.735,E2 27255.735} C_VEL
LIN {X 0,Y 576.418,Z 732.554,A -85,B 0,C 180,E1 27253.939,E2 27253.939} C_VEL
LIN {X 0,Y 576.65,Z 717.952,A -85,B 0,C 180,E1 27252.231,E2 27252.231} C_VEL
LIN {X 0,Y 576.931,Z 702.17,A -85,B 0,C 180,E1 27250.669,E2 27250.669} C_VEL
LIN {X 0,Y 577.235,Z 685.35,A -85,B 0,C 180,E1 27249.259,E2 27249.259} C_VEL
LIN {X 0,Y 577.543,Z 668.135,A -85,B 0,C 180,E1 27248.04,E2 27248.04} C_VEL
LIN {X 0,Y 577.869,Z 649.262,A -85,B 0,C 180,E1 27246.926,E2 27246.926} C_VEL
LIN {X 0,Y 578.193,Z 629.24,A -85,B 0,C 180,E1 27245.967,E2 27245.967} C_VEL
LIN {X 0,Y 578.494,Z 609.339,A -85,B 0,C 180,E1 27245.219,E2 27245.219} C_VEL
LIN {X 0,Y 578.736,Z 589.022,A -85,B 0,C 180,E1 27244.65,E2 27244.65} C_VEL
LIN {X 0,Y 578.868,Z 568.031,A -85,B 0,C 180,E1 27244.262,E2 27244.262} C_VEL
LIN {X 0,Y 579.622,Z 333.536,A -85,B 0,C 180,E1 27241.091,E2 27241.091} C_VEL
LIN {X 0,Y 579.439,Z 319.158,A -85,B 0,C 180,E1 27240.881,E2 27240.881} C_VEL
LIN {X 0,Y 578.776,Z 314.495,A -85,B 0,C 180,E1 27240.739,E2 27240.739} C_VEL
LIN {X 0,Y 579.284,Z 273.474,A -85,B 0,C 180,E1 27237.98,E2 27237.98} C_VEL
LIN {X 0,Y 576.188,Z 264.941,A -85,B 0,C 180,E1 27237.152,E2 27237.152} C_VEL
LIN {X 0,Y 576.132,Z 264.717,A -85,B 0,C 180,E1 27233.961,E2 27233.961} C_VEL
LIN {X 0,Y 576.128,Z 264.72,A -85,B 0,C 180,E1 27230.56,E2 27230.56} C_VEL
LIN {X 0,Y 576.16,Z 264.716,A -85,B 0,C 180,E1 27227.375,E2 27227.375} C_VEL
LIN {X 0,Y 576.115,Z 264.718,A -85,B 0,C 180,E1 27224.211,E2 27224.211} C_VEL
LIN {X 0,Y 576.161,Z 264.72,A -85,B 0,C 180,E1 27220.983,E2 27220.983} C_VEL
LIN {X 0,Y 576.126,Z 264.717,A -85,B 0,C 180,E1 27217.779,E2 27217.779} C_VEL
LIN {X 0,Y 576.115,Z 264.722,A -85,B 0,C 180,E1 27214.456,E2 27214.456} C_VEL
LIN {X 0,Y 576.16,Z 264.709,A -85,B 0,C 180,E1 27211.257,E2 27211.257} C_VEL
LIN {X 0,Y 576.164,Z 265.039,A -85,B 0,C 180,E1 27210.532,E2 27210.532} C_VEL
LIN {X 0,Y 578.615,Z 273.057,A -85,B 0,C 180,E1 27209.732,E2 27209.732} C_VEL
LIN {X 0,Y 578.061,Z 313.726,A -85,B 0,C 180,E1 27206.588,E2 27206.588} C_VEL
LIN {X 0,Y 577.847,Z 342.642,A -85,B 0,C 180,E1 27204.427,E2 27204.427} C_VEL
LIN {X 0,Y 578.574,Z 348.669,A -85,B 0,C 180,E1 27204.309,E2 27204.309} C_VEL
LIN {X 0,Y 577.985,Z 559.915,A -85,B 0,C 180,E1 27201.514,E2 27201.514} C_VEL
LIN {X 0,Y 577.826,Z 579.635,A -85,B 0,C 180,E1 27201.058,E2 27201.058} C_VEL
LIN {X 0,Y 577.628,Z 598.179,A -85,B 0,C 180,E1 27200.44,E2 27200.44} C_VEL
LIN {X 0,Y 577.387,Z 616.468,A -85,B 0,C 180,E1 27199.63,E2 27199.63} C_VEL
LIN {X 0,Y 577.127,Z 634.544,A -85,B 0,C 180,E1 27198.617,E2 27198.617} C_VEL
LIN {X 0,Y 576.872,Z 650.743,A -85,B 0,C 180,E1 27197.5,E2 27197.5} C_VEL
LIN {X 0,Y 576.626,Z 666.249,A -85,B 0,C 180,E1 27196.21,E2 27196.21} C_VEL
LIN {X 0,Y 576.407,Z 680.631,A -85,B 0,C 180,E1 27194.773,E2 27194.773} C_VEL
LIN {X 0,Y 576.239,Z 693.478,A -85,B 0,C 180,E1 27193.239,E2 27193.239} C_VEL
LIN {X 0,Y 576.105,Z 704.801,A -85,B 0,C 180,E1 27191.614,E2 27191.614} C_VEL
LIN {X 0,Y 576.012,Z 714.642,A -85,B 0,C 180,E1 27189.895,E2 27189.895} C_VEL
LIN {X 0,Y 575.955,Z 722.965,A -85,B 0,C 180,E1 27188.083,E2 27188.083} C_VEL
LIN {X 0,Y 575.926,Z 729.708,A -85,B 0,C 180,E1 27186.179,E2 27186.179} C_VEL
LIN {X 0,Y 575.91,Z 734.537,A -85,B 0,C 180,E1 27184.281,E2 27184.281} C_VEL
LIN {X 0,Y 575.914,Z 737.569,A -85,B 0,C 180,E1 27182.388,E2 27182.388} C_VEL
LIN {X 0,Y 575.908,Z 738.885,A -85,B 0,C 180,E1 27180.497,E2 27180.497} C_VEL
LIN {X 0,Y 575.912,Z 738.465,A -85,B 0,C 180,E1 27178.507,E2 27178.507} C_VEL
LIN {X 0,Y 575.913,Z 736.334,A -85,B 0,C 180,E1 27176.616,E2 27176.616} C_VEL
LIN {X 0,Y 575.92,Z 732.453,A -85,B 0,C 180,E1 27174.72,E2 27174.72} C_VEL
LIN {X 0,Y 575.944,Z 726.725,A -85,B 0,C 180,E1 27172.819,E2 27172.819} C_VEL
LIN {X 0,Y 575.985,Z 719.001,A -85,B 0,C 180,E1 27170.911,E2 27170.911} C_VEL
LIN {X 0,Y 576.061,Z 709.623,A -85,B 0,C 180,E1 27169.094,E2 27169.094} C_VEL
LIN {X 0,Y 576.172,Z 698.969,A -85,B 0,C 180,E1 27167.42,E2 27167.42} C_VEL
LIN {X 0,Y 576.325,Z 686.817,A -85,B 0,C 180,E1 27165.84,E2 27165.84} C_VEL
LIN {X 0,Y 576.462,Z 677.121,A -85,B 0,C 180,E1 27164.76,E2 27164.76} C_VEL
LIN {X 0,Y 575.534,Z 671.912,A -85,B 0,C 180,E1 27164.203,E2 27164.203} C_VEL
LIN {X 0,Y 569.928,Z 658.431,A -85,B 0,C 180,E1 27162.81,E2 27162.81} C_VEL
LIN {X 0,Y 569.093,Z 652.545,A -85,B 0,C 180,E1 27162.305,E2 27162.305} C_VEL
LIN {X 0,Y 569.414,Z 636.354,A -85,B 0,C 180,E1 27161.149,E2 27161.149} C_VEL
LIN {X 0,Y 569.729,Z 619.186,A -85,B 0,C 180,E1 27160.148,E2 27160.148} C_VEL
LIN {X 0,Y 570.031,Z 600.967,A -85,B 0,C 180,E1 27159.302,E2 27159.302} C_VEL
LIN {X 0,Y 570.301,Z 582.037,A -85,B 0,C 180,E1 27158.633,E2 27158.633} C_VEL
LIN {X 0,Y 570.505,Z 562.731,A -85,B 0,C 180,E1 27158.155,E2 27158.155} C_VEL
LIN {X 0,Y 570.667,Z 532.892,A -85,B 0,C 180,E1 27157.718,E2 27157.718} C_VEL
LIN {X 0,Y 571.13,Z 347.18,A -85,B 0,C 180,E1 27155.243,E2 27155.243} C_VEL
LIN {X 0,Y 570.292,Z 342.045,A -85,B 0,C 180,E1 27155.116,E2 27155.116} C_VEL
LIN {X 0,Y 570.913,Z 299.398,A -85,B 0,C 180,E1 27151.836,E2 27151.836} C_VEL
LIN {X 0,Y 571.231,Z 275.144,A -85,B 0,C 180,E1 27149.922,E2 27149.922} C_VEL
LIN {X 0,Y 568.25,Z 265.922,A -85,B 0,C 180,E1 27148.966,E2 27148.966} C_VEL
LIN {X 0,Y 568.171,Z 265.688,A -85,B 0,C 180,E1 27145.727,E2 27145.727} C_VEL
LIN {X 0,Y 568.213,Z 265.703,A -85,B 0,C 180,E1 27142.494,E2 27142.494} C_VEL
LIN {X 0,Y 568.222,Z 265.708,A -85,B 0,C 180,E1 27139.17,E2 27139.17} C_VEL
LIN {X 0,Y 568.192,Z 265.705,A -85,B 0,C 180,E1 27135.888,E2 27135.888} C_VEL
LIN {X 0,Y 568.216,Z 265.702,A -85,B 0,C 180,E1 27132.647,E2 27132.647} C_VEL
LIN {X 0,Y 568.216,Z 265.708,A -85,B 0,C 180,E1 27129.263,E2 27129.263} C_VEL
LIN {X 0,Y 568.207,Z 265.704,A -85,B 0,C 180,E1 27125.957,E2 27125.957} C_VEL
LIN {X 0,Y 568.201,Z 265.702,A -85,B 0,C 180,E1 27122.7,E2 27122.7} C_VEL
LIN {X 0,Y 568.198,Z 265.706,A -85,B 0,C 180,E1 27119.289,E2 27119.289} C_VEL
LIN {X 0,Y 568.219,Z 265.705,A -85,B 0,C 180,E1 27115.987,E2 27115.987} C_VEL
LIN {X 0,Y 568.181,Z 265.705,A -85,B 0,C 180,E1 27112.762,E2 27112.762} C_VEL
LIN {X 0,Y 568.182,Z 265.708,A -85,B 0,C 180,E1 27109.398,E2 27109.398} C_VEL
LIN {X 0,Y 568.211,Z 265.706,A -85,B 0,C 180,E1 27106.248,E2 27106.248} C_VEL
LIN {X 0,Y 568.153,Z 265.708,A -85,B 0,C 180,E1 27103.123,E2 27103.123} C_VEL
LIN {X 0,Y 568.205,Z 265.697,A -85,B 0,C 180,E1 27099.931,E2 27099.931} C_VEL
LIN {X 0,Y 568.208,Z 265.914,A -85,B 0,C 180,E1 27097.763,E2 27097.763} C_VEL
LIN {X 0,Y 570.584,Z 274.579,A -85,B 0,C 180,E1 27096.946,E2 27096.946} C_VEL
LIN {X 0,Y 570.58,Z 314.764,A -85,B 0,C 180,E1 27093.869,E2 27093.869} C_VEL
LIN {X 0,Y 570.343,Z 356.327,A -85,B 0,C 180,E1 27090.704,E2 27090.704} C_VEL
LIN {X 0,Y 569.832,Z 396.228,A -85,B 0,C 180,E1 27087.638,E2 27087.638} C_VEL
LIN {X 0,Y 569.309,Z 440.162,A -85,B 0,C 180,E1 27084.306,E2 27084.306} C_VEL
LIN {X 0,Y 569.015,Z 472.31,A -85,B 0,C 180,E1 27081.92,E2 27081.92} C_VEL
LIN {X 0,Y 569.493,Z 479.62,A -85,B 0,C 180,E1 27081.797,E2 27081.797} C_VEL
LIN {X 0,Y 569.149,Z 615.458,A -85,B 0,C 180,E1 27080.033,E2 27080.033} C_VEL
LIN {X 0,Y 569.049,Z 632.104,A -85,B 0,C 180,E1 27079.616,E2 27079.616} C_VEL
LIN {X 0,Y 568.896,Z 647.047,A -85,B 0,C 180,E1 27079.059,E2 27079.059} C_VEL
LIN {X 0,Y 568.703,Z 662.249,A -85,B 0,C 180,E1 27078.29,E2 27078.29} C_VEL
LIN {X 0,Y 568.515,Z 676.52,A -85,B 0,C 180,E1 27077.353,E2 27077.353} C_VEL
LIN {X 0,Y 568.34,Z 689.626,A -85,B 0,C 180,E1 27076.262,E2 27076.262} C_VEL
LIN {X 0,Y 568.187,Z 701.677,A -85,B 0,C 180,E1 27075.01,E2 27075.01} C_VEL
LIN {X 0,Y 568.07,Z 712.106,A -85,B 0,C 180,E1 27073.645,E2 27073.645} C_VEL
LIN {X 0,Y 567.993,Z 721.041,A -85,B 0,C 180,E1 27072.165,E2 27072.165} C_VEL
LIN {X 0,Y 567.945,Z 727.94,A -85,B 0,C 180,E1 27070.67,E2 27070.67} C_VEL
LIN {X 0,Y 567.926,Z 733.391,A -85,B 0,C 180,E1 27069.061,E2 27069.061} C_VEL
LIN {X 0,Y 567.916,Z 736.958,A -85,B 0,C 180,E1 27067.432,E2 27067.432} C_VEL
LIN {X 0,Y 567.918,Z 738.756,A -85,B 0,C 180,E1 27065.781,E2 27065.781} C_VEL
LIN {X 0,Y 567.915,Z 738.818,A -85,B 0,C 180,E1 27064.225,E2 27064.225} C_VEL
LIN {X 0,Y 567.916,Z 737.039,A -85,B 0,C 180,E1 27062.532,E2 27062.532} C_VEL
LIN {X 0,Y 567.923,Z 733.621,A -85,B 0,C 180,E1 27060.929,E2 27060.929} C_VEL
LIN {X 0,Y 567.945,Z 728.188,A -85,B 0,C 180,E1 27059.302,E2 27059.302} C_VEL
LIN {X 0,Y 567.992,Z 721.158,A -85,B 0,C 180,E1 27057.767,E2 27057.767} C_VEL
LIN {X 0,Y 568.064,Z 712.542,A -85,B 0,C 180,E1 27056.33,E2 27056.33} C_VEL
LIN {X 0,Y 568.187,Z 701.789,A -85,B 0,C 180,E1 27054.914,E2 27054.914} C_VEL
LIN {X 0,Y 568.334,Z 690.011,A -85,B 0,C 180,E1 27053.684,E2 27053.684} C_VEL
LIN {X 0,Y 568.511,Z 677.153,A -85,B 0,C 180,E1 27052.603,E2 27052.603} C_VEL
LIN {X 0,Y 568.697,Z 662.595,A -85,B 0,C 180,E1 27051.64,E2 27051.64} C_VEL
LIN {X 0,Y 568.883,Z 647.742,A -85,B 0,C 180,E1 27050.88,E2 27050.88} C_VEL
LIN {X 0,Y 569.05,Z 631.274,A -85,B 0,C 180,E1 27050.267,E2 27050.267} C_VEL
LIN {X 0,Y 569.137,Z 614.862,A -85,B 0,C 180,E1 27049.866,E2 27049.866} C_VEL
LIN {X 0,Y 569.279,Z 474.786,A -85,B 0,C 180,E1 27048.044,E2 27048.044} C_VEL
LIN {X 0,Y 568.985,Z 472.015,A -85,B 0,C 180,E1 27047.972,E2 27047.972} C_VEL
LIN {X 0,Y 569.413,Z 430.843,A -85,B 0,C 180,E1 27044.902,E2 27044.902} C_VEL
LIN {X 0,Y 569.893,Z 388.518,A -85,B 0,C 180,E1 27041.679,E2 27041.679} C_VEL
LIN {X 0,Y 570.364,Z 352.171,A -85,B 0,C 180,E1 27038.894,E2 27038.894} C_VEL
LIN {X 0,Y 570.457,Z 309.748,A -85,B 0,C 180,E1 27035.709,E2 27035.709} C_VEL
LIN {X 0,Y 570.392,Z 279.968,A -85,B 0,C 180,E1 27033.45,E2 27033.45} C_VEL
LIN {X 0,Y 570.083,Z 272.371,A -85,B 0,C 180,E1 27032.871,E2 27032.871} C_VEL
LIN {X 0,Y 568.225,Z 266.024,A -85,B 0,C 180,E1 27032.28,E2 27032.28} C_VEL
LIN {X 0,Y 568.222,Z 265.707,A -85,B 0,C 180,E1 27031.611,E2 27031.611} C_VEL
LIN {X 0,Y 568.171,Z 265.708,A -85,B 0,C 180,E1 27028.484,E2 27028.484} C_VEL
LIN {X 0,Y 568.211,Z 265.705,A -85,B 0,C 180,E1 27025.204,E2 27025.204} C_VEL
LIN {X 0,Y 568.195,Z 265.71,A -85,B 0,C 180,E1 27021.977,E2 27021.977} C_VEL
LIN {X 0,Y 568.178,Z 265.704,A -85,B 0,C 180,E1 27018.68,E2 27018.68} C_VEL
LIN {X 0,Y 568.222,Z 265.706,A -85,B 0,C 180,E1 27015.514,E2 27015.514} C_VEL
LIN {X 0,Y 568.175,Z 265.707,A -85,B 0,C 180,E1 27012.295,E2 27012.295} C_VEL
LIN {X 0,Y 568.212,Z 265.702,A -85,B 0,C 180,E1 27009.011,E2 27009.011} C_VEL
LIN {X 0,Y 568.204,Z 265.709,A -85,B 0,C 180,E1 27005.757,E2 27005.757} C_VEL
LIN {X 0,Y 568.177,Z 265.705,A -85,B 0,C 180,E1 27002.421,E2 27002.421} C_VEL
LIN {X 0,Y 568.22,Z 265.704,A -85,B 0,C 180,E1 26999.194,E2 26999.194} C_VEL
LIN {X 0,Y 568.183,Z 265.707,A -85,B 0,C 180,E1 26995.964,E2 26995.964} C_VEL
LIN {X 0,Y 568.195,Z 265.702,A -85,B 0,C 180,E1 26992.62,E2 26992.62} C_VEL
LIN {X 0,Y 568.219,Z 265.708,A -85,B 0,C 180,E1 26989.353,E2 26989.353} C_VEL
LIN {X 0,Y 568.179,Z 265.705,A -85,B 0,C 180,E1 26986.153,E2 26986.153} C_VEL
LIN {X 0,Y 568.221,Z 265.702,A -85,B 0,C 180,E1 26982.911,E2 26982.911} C_VEL
LIN {X 0,Y 568.199,Z 265.708,A -85,B 0,C 180,E1 26979.61,E2 26979.61} C_VEL
LIN {X 0,Y 568.184,Z 265.704,A -85,B 0,C 180,E1 26976.236,E2 26976.236} C_VEL
LIN {X 0,Y 568.219,Z 265.704,A -85,B 0,C 180,E1 26973.001,E2 26973.001} C_VEL
LIN {X 0,Y 568.186,Z 265.706,A -85,B 0,C 180,E1 26969.769,E2 26969.769} C_VEL
LIN {X 0,Y 568.207,Z 265.701,A -85,B 0,C 180,E1 26966.459,E2 26966.459} C_VEL
LIN {X 0,Y 568.22,Z 265.708,A -85,B 0,C 180,E1 26963.128,E2 26963.128} C_VEL
LIN {X 0,Y 568.184,Z 265.705,A -85,B 0,C 180,E1 26959.905,E2 26959.905} C_VEL
LIN {X 0,Y 568.22,Z 265.703,A -85,B 0,C 180,E1 26956.61,E2 26956.61} C_VEL
LIN {X 0,Y 568.212,Z 265.709,A -85,B 0,C 180,E1 26953.24,E2 26953.24} C_VEL
LIN {X 0,Y 568.188,Z 265.705,A -85,B 0,C 180,E1 26949.962,E2 26949.962} C_VEL
LIN {X 0,Y 568.214,Z 265.69,A -85,B 0,C 180,E1 26946.745,E2 26946.745} C_VEL
LIN {X 0,Y 568.191,Z 265.706,A -85,B 0,C 180,E1 26943.477,E2 26943.477} C_VEL
LIN {X 0,Y 568.308,Z 266.324,A -85,B 0,C 180,E1 26943.238,E2 26943.238} C_VEL
LIN {X 0,Y 572.185,Z 277.197,A -85,B 0,C 180,E1 26942.204,E2 26942.204} C_VEL
LIN {X 0,Y 571.647,Z 315.823,A -85,B 0,C 180,E1 26939.605,E2 26939.605} C_VEL
LIN {X 0,Y 572.659,Z 323.284,A -85,B 0,C 180,E1 26939.439,E2 26939.439} C_VEL
LIN {X 0,Y 571.734,Z 552.304,A -85,B 0,C 180,E1 26936.302,E2 26936.302} C_VEL
LIN {X 0,Y 571.544,Z 581.049,A -85,B 0,C 180,E1 26935.864,E2 26935.864} C_VEL
LIN {X 0,Y 571.308,Z 601.407,A -85,B 0,C 180,E1 26935.368,E2 26935.368} C_VEL
LIN {X 0,Y 570.995,Z 621.202,A -85,B 0,C 180,E1 26934.695,E2 26934.695} C_VEL
LIN {X 0,Y 570.609,Z 639.891,A -85,B 0,C 180,E1 26933.875,E2 26933.875} C_VEL
LIN {X 0,Y 570.21,Z 658.766,A -85,B 0,C 180,E1 26932.853,E2 26932.853} C_VEL
LIN {X 0,Y 569.785,Z 677.478,A -85,B 0,C 180,E1 26931.622,E2 26931.622} C_VEL
LIN {X 0,Y 569.391,Z 694.356,A -85,B 0,C 180,E1 26930.296,E2 26930.296} C_VEL
LIN {X 0,Y 569.023,Z 710.417,A -85,B 0,C 180,E1 26928.809,E2 26928.809} C_VEL
LIN {X 0,Y 568.698,Z 725.365,A -85,B 0,C 180,E1 26927.178,E2 26927.178} C_VEL
LIN {X 0,Y 568.433,Z 739.137,A -85,B 0,C 180,E1 26925.402,E2 26925.402} C_VEL
LIN {X 0,Y 568.219,Z 751.298,A -85,B 0,C 180,E1 26923.533,E2 26923.533} C_VEL
LIN {X 0,Y 568.077,Z 761.373,A -85,B 0,C 180,E1 26921.677,E2 26921.677} C_VEL
LIN {X 0,Y 567.993,Z 770.289,A -85,B 0,C 180,E1 26919.672,E2 26919.672} C_VEL
LIN {X 0,Y 567.945,Z 777.475,A -85,B 0,C 180,E1 26917.628,E2 26917.628} C_VEL
LIN {X 0,Y 567.92,Z 782.732,A -85,B 0,C 180,E1 26915.657,E2 26915.657} C_VEL
LIN {X 0,Y 567.908,Z 786.402,A -85,B 0,C 180,E1 26913.633,E2 26913.633} C_VEL
LIN {X 0,Y 567.902,Z 788.441,A -85,B 0,C 180,E1 26911.613,E2 26911.613} C_VEL
LIN {X 0,Y 567.9,Z 788.895,A -85,B 0,C 180,E1 26909.495,E2 26909.495} C_VEL
LIN {X 0,Y 567.907,Z 787.727,A -85,B 0,C 180,E1 26907.476,E2 26907.476} C_VEL
LIN {X 0,Y 567.913,Z 784.97,A -85,B 0,C 180,E1 26905.455,E2 26905.455} C_VEL
LIN {X 0,Y 567.931,Z 780.48,A -85,B 0,C 180,E1 26903.428,E2 26903.428} C_VEL
LIN {X 0,Y 567.969,Z 774.262,A -85,B 0,C 180,E1 26901.393,E2 26901.393} C_VEL
LIN {X 0,Y 568.028,Z 766.175,A -85,B 0,C 180,E1 26899.348,E2 26899.348} C_VEL
LIN {X 0,Y 568.143,Z 756.561,A -85,B 0,C 180,E1 26897.394,E2 26897.394} C_VEL
LIN {X 0,Y 568.325,Z 745.488,A -85,B 0,C 180,E1 26895.532,E2 26895.532} C_VEL
LIN {X 0,Y 568.551,Z 732.933,A -85,B 0,C 180,E1 26893.762,E2 26893.762} C_VEL
LIN {X 0,Y 568.832,Z 718.879,A -85,B 0,C 180,E1 26892.084,E2 26892.084} C_VEL
LIN {X 0,Y 569.169,Z 703.833,A -85,B 0,C 180,E1 26890.555,E2 26890.555} C_VEL
LIN {X 0,Y 569.551,Z 687.283,A -85,B 0,C 180,E1 26889.122,E2 26889.122} C_VEL
LIN {X 0,Y 569.976,Z 668.941,A -85,B 0,C 180,E1 26887.787,E2 26887.787} C_VEL
LIN {X 0,Y 570.388,Z 650.263,A -85,B 0,C 180,E1 26886.66,E2 26886.66} C_VEL
LIN {X 0,Y 570.784,Z 631.791,A -85,B 0,C 180,E1 26885.745,E2 26885.745} C_VEL
LIN {X 0,Y 571.16,Z 611.854,A -85,B 0,C 180,E1 26884.962,E2 26884.962} C_VEL
LIN {X 0,Y 571.428,Z 591.582,A -85,B 0,C 180,E1 26884.37,E2 26884.37} C_VEL
LIN {X 0,Y 571.638,Z 571.154,A -85,B 0,C 180,E1 26883.963,E2 26883.963} C_VEL
LIN {X 0,Y 572.618,Z 333.536,A -85,B 0,C 180,E1 26880.703,E2 26880.703} C_VEL
LIN {X 0,Y 572.442,Z 320.457,A -85,B 0,C 180,E1 26880.509,E2 26880.509} C_VEL
LIN {X 0,Y 571.564,Z 314.836,A -85,B 0,C 180,E1 26880.354,E2 26880.354} C_VEL
LIN {X 0,Y 572.165,Z 276.654,A -85,B 0,C 180,E1 26877.756,E2 26877.756} C_VEL
LIN {X 0,Y 568.247,Z 266.023,A -85,B 0,C 180,E1 26876.721,E2 26876.721} C_VEL
LIN {X 0,Y 568.203,Z 265.709,A -85,B 0,C 180,E1 26875.851,E2 26875.851} C_VEL
LIN {X 0,Y 568.186,Z 265.71,A -85,B 0,C 180,E1 26872.491,E2 26872.491} C_VEL
LIN {X 0,Y 568.221,Z 265.707,A -85,B 0,C 180,E1 26869.244,E2 26869.244} C_VEL
LIN {X 0,Y 568.185,Z 265.706,A -85,B 0,C 180,E1 26865.964,E2 26865.964} C_VEL
LIN {X 0,Y 568.192,Z 265.71,A -85,B 0,C 180,E1 26862.644,E2 26862.644} C_VEL
LIN {X 0,Y 568.224,Z 265.704,A -85,B 0,C 180,E1 26859.423,E2 26859.423} C_VEL
LIN {X 0,Y 568.171,Z 265.709,A -85,B 0,C 180,E1 26856.248,E2 26856.248} C_VEL
LIN {X 0,Y 568.219,Z 265.709,A -85,B 0,C 180,E1 26853.058,E2 26853.058} C_VEL
LIN {X 0,Y 568.251,Z 265.927,A -85,B 0,C 180,E1 26850.945,E2 26850.945} C_VEL
LIN {X 0,Y 571.301,Z 275.947,A -85,B 0,C 180,E1 26849.92,E2 26849.92} C_VEL
LIN {X 0,Y 570.614,Z 317.064,A -85,B 0,C 180,E1 26846.703,E2 26846.703} C_VEL
LIN {X 0,Y 570.322,Z 342.297,A -85,B 0,C 180,E1 26844.785,E2 26844.785} C_VEL
LIN {X 0,Y 571.283,Z 349.569,A -85,B 0,C 180,E1 26844.628,E2 26844.628} C_VEL
LIN {X 0,Y 570.541,Z 559.942,A -85,B 0,C 180,E1 26841.809,E2 26841.809} C_VEL
LIN {X 0,Y 570.341,Z 579.649,A -85,B 0,C 180,E1 26841.348,E2 26841.348} C_VEL
LIN {X 0,Y 570.092,Z 598.197,A -85,B 0,C 180,E1 26840.722,E2 26840.722} C_VEL
LIN {X 0,Y 569.786,Z 616.477,A -85,B 0,C 180,E1 26839.903,E2 26839.903} C_VEL
LIN {X 0,Y 569.463,Z 634.177,A -85,B 0,C 180,E1 26838.901,E2 26838.901} C_VEL
LIN {X 0,Y 569.137,Z 650.753,A -85,B 0,C 180,E1 26837.746,E2 26837.746} C_VEL
LIN {X 0,Y 568.827,Z 666.254,A -85,B 0,C 180,E1 26836.439,E2 26836.439} C_VEL
LIN {X 0,Y 568.552,Z 680.636,A -85,B 0,C 180,E1 26834.982,E2 26834.982} C_VEL
LIN {X 0,Y 568.336,Z 693.477,A -85,B 0,C 180,E1 26833.428,E2 26833.428} C_VEL
LIN {X 0,Y 568.164,Z 704.809,A -85,B 0,C 180,E1 26831.779,E2 26831.779} C_VEL
LIN {X 0,Y 568.047,Z 714.647,A -85,B 0,C 180,E1 26830.035,E2 26830.035} C_VEL
LIN {X 0,Y 567.968,Z 722.967,A -85,B 0,C 180,E1 26828.198,E2 26828.198} C_VEL
LIN {X 0,Y 567.933,Z 729.712,A -85,B 0,C 180,E1 26826.266,E2 26826.266} C_VEL
LIN {X 0,Y 567.911,Z 734.541,A -85,B 0,C 180,E1 26824.341,E2 26824.341} C_VEL
LIN {X 0,Y 567.913,Z 737.572,A -85,B 0,C 180,E1 26822.421,E2 26822.421} C_VEL
LIN {X 0,Y 567.908,Z 738.885,A -85,B 0,C 180,E1 26820.504,E2 26820.504} C_VEL
LIN {X 0,Y 567.912,Z 738.466,A -85,B 0,C 180,E1 26818.486,E2 26818.486} C_VEL
LIN {X 0,Y 567.911,Z 736.336,A -85,B 0,C 180,E1 26816.568,E2 26816.568} C_VEL
LIN {X 0,Y 567.922,Z 732.454,A -85,B 0,C 180,E1 26814.646,E2 26814.646} C_VEL
LIN {X 0,Y 567.95,Z 726.724,A -85,B 0,C 180,E1 26812.718,E2 26812.718} C_VEL
LIN {X 0,Y 568.009,Z 718.999,A -85,B 0,C 180,E1 26810.782,E2 26810.782} C_VEL
LIN {X 0,Y 568.11,Z 709.622,A -85,B 0,C 180,E1 26808.94,E2 26808.94} C_VEL
LIN {X 0,Y 568.258,Z 698.617,A -85,B 0,C 180,E1 26807.191,E2 26807.191} C_VEL
LIN {X 0,Y 568.444,Z 686.814,A -85,B 0,C 180,E1 26805.64,E2 26805.64} C_VEL
LIN {X 0,Y 568.684,Z 673.62,A -85,B 0,C 180,E1 26804.185,E2 26804.185} C_VEL
LIN {X 0,Y 568.971,Z 658.977,A -85,B 0,C 180,E1 26802.828,E2 26802.828} C_VEL
LIN {X 0,Y 569.093,Z 652.545,A -85,B 0,C 180,E1 26802.305,E2 26802.305} C_VEL
LIN {X 0,Y 568.272,Z 646.543,A -85,B 0,C 180,E1 26801.815,E2 26801.815} C_VEL
LIN {X 0,Y 562.847,Z 631.343,A -85,B 0,C 180,E1 26800.598,E2 26800.598} C_VEL
LIN {X 0,Y 562.015,Z 624.834,A -85,B 0,C 180,E1 26800.178,E2 26800.178} C_VEL
LIN {X 0,Y 562.403,Z 607.236,A -85,B 0,C 180,E1 26799.28,E2 26799.28} C_VEL
LIN {X 0,Y 562.74,Z 588.423,A -85,B 0,C 180,E1 26798.54,E2 26798.54} C_VEL
LIN {X 0,Y 563.017,Z 568.721,A -85,B 0,C 180,E1 26797.979,E2 26797.979} C_VEL
LIN {X 0,Y 563.199,Z 548.932,A -85,B 0,C 180,E1 26797.624,E2 26797.624} C_VEL
LIN {X 0,Y 563.871,Z 348.428,A -85,B 0,C 180,E1 26794.92,E2 26794.92} C_VEL
LIN {X 0,Y 562.822,Z 342.045,A -85,B 0,C 180,E1 26794.763,E2 26794.763} C_VEL
LIN {X 0,Y 563.583,Z 299.244,A -85,B 0,C 180,E1 26791.425,E2 26791.425} C_VEL
LIN {X 0,Y 563.903,Z 277.869,A -85,B 0,C 180,E1 26789.713,E2 26789.713} C_VEL
LIN {X 0,Y 560.31,Z 266.962,A -85,B 0,C 180,E1 26788.568,E2 26788.568} C_VEL
LIN {X 0,Y 560.233,Z 266.674,A -85,B 0,C 180,E1 26785.669,E2 26785.669} C_VEL
LIN {X 0,Y 560.264,Z 266.693,A -85,B 0,C 180,E1 26782.385,E2 26782.385} C_VEL
LIN {X 0,Y 560.282,Z 266.696,A -85,B 0,C 180,E1 26779.085,E2 26779.085} C_VEL
LIN {X 0,Y 560.255,Z 266.695,A -85,B 0,C 180,E1 26775.749,E2 26775.749} C_VEL
LIN {X 0,Y 560.276,Z 266.69,A -85,B 0,C 180,E1 26772.368,E2 26772.368} C_VEL
LIN {X 0,Y 560.269,Z 266.695,A -85,B 0,C 180,E1 26769.048,E2 26769.048} C_VEL
LIN {X 0,Y 560.273,Z 266.696,A -85,B 0,C 180,E1 26765.702,E2 26765.702} C_VEL
LIN {X 0,Y 560.279,Z 266.689,A -85,B 0,C 180,E1 26762.37,E2 26762.37} C_VEL
LIN {X 0,Y 560.25,Z 266.692,A -85,B 0,C 180,E1 26759.015,E2 26759.015} C_VEL
LIN {X 0,Y 560.279,Z 266.694,A -85,B 0,C 180,E1 26755.681,E2 26755.681} C_VEL
LIN {X 0,Y 560.272,Z 266.692,A -85,B 0,C 180,E1 26752.342,E2 26752.342} C_VEL
LIN {X 0,Y 560.23,Z 266.696,A -85,B 0,C 180,E1 26749.064,E2 26749.064} C_VEL
LIN {X 0,Y 560.275,Z 266.694,A -85,B 0,C 180,E1 26745.846,E2 26745.846} C_VEL
LIN {X 0,Y 560.225,Z 266.696,A -85,B 0,C 180,E1 26742.682,E2 26742.682} C_VEL
LIN {X 0,Y 560.209,Z 266.692,A -85,B 0,C 180,E1 26739.348,E2 26739.348} C_VEL
LIN {X 0,Y 560.309,Z 266.955,A -85,B 0,C 180,E1 26738.079,E2 26738.079} C_VEL
LIN {X 0,Y 563.12,Z 276.791,A -85,B 0,C 180,E1 26737.141,E2 26737.141} C_VEL
LIN {X 0,Y 563.06,Z 315.928,A -85,B 0,C 180,E1 26734.125,E2 26734.125} C_VEL
LIN {X 0,Y 562.759,Z 357.058,A -85,B 0,C 180,E1 26730.968,E2 26730.968} C_VEL
LIN {X 0,Y 562.252,Z 395.027,A -85,B 0,C 180,E1 26728.048,E2 26728.048} C_VEL
LIN {X 0,Y 561.645,Z 439.417,A -85,B 0,C 180,E1 26724.638,E2 26724.638} C_VEL
LIN {X 0,Y 561.272,Z 472.478,A -85,B 0,C 180,E1 26722.156,E2 26722.156} C_VEL
LIN {X 0,Y 561.834,Z 480.229,A -85,B 0,C 180,E1 26722.025,E2 26722.025} C_VEL
LIN {X 0,Y 561.421,Z 615.352,A -85,B 0,C 180,E1 26720.248,E2 26720.248} C_VEL
LIN {X 0,Y 561.296,Z 631.802,A -85,B 0,C 180,E1 26719.833,E2 26719.833} C_VEL
LIN {X 0,Y 561.1,Z 648.005,A -85,B 0,C 180,E1 26719.217,E2 26719.217} C_VEL
LIN {X 0,Y 560.866,Z 663.048,A -85,B 0,C 180,E1 26718.432,E2 26718.432} C_VEL
LIN {X 0,Y 560.64,Z 677.243,A -85,B 0,C 180,E1 26717.476,E2 26717.476} C_VEL
LIN {X 0,Y 560.42,Z 690.634,A -85,B 0,C 180,E1 26716.327,E2 26716.327} C_VEL
LIN {X 0,Y 560.245,Z 702.045,A -85,B 0,C 180,E1 26715.11,E2 26715.11} C_VEL
LIN {X 0,Y 560.103,Z 712.396,A -85,B 0,C 180,E1 26713.725,E2 26713.725} C_VEL
LIN {X 0,Y 560.008,Z 721.264,A -85,B 0,C 180,E1 26712.225,E2 26712.225} C_VEL
LIN {X 0,Y 559.948,Z 728.518,A -85,B 0,C 180,E1 26710.604,E2 26710.604} C_VEL
LIN {X 0,Y 559.928,Z 733.575,A -85,B 0,C 180,E1 26709.055,E2 26709.055} C_VEL
LIN {X 0,Y 559.916,Z 737.056,A -85,B 0,C 180,E1 26707.403,E2 26707.403} C_VEL
LIN {X 0,Y 559.918,Z 738.783,A -85,B 0,C 180,E1 26705.752,E2 26705.752} C_VEL
LIN {X 0,Y 559.915,Z 738.784,A -85,B 0,C 180,E1 26704.161,E2 26704.161} C_VEL
LIN {X 0,Y 559.916,Z 736.969,A -85,B 0,C 180,E1 26702.453,E2 26702.453} C_VEL
LIN {X 0,Y 559.929,Z 733.494,A -85,B 0,C 180,E1 26700.826,E2 26700.826} C_VEL
LIN {X 0,Y 559.953,Z 728.002,A -85,B 0,C 180,E1 26699.173,E2 26699.173} C_VEL
LIN {X 0,Y 560.011,Z 720.905,A -85,B 0,C 180,E1 26697.615,E2 26697.615} C_VEL
LIN {X 0,Y 560.11,Z 711.882,A -85,B 0,C 180,E1 26696.108,E2 26696.108} C_VEL
LIN {X 0,Y 560.245,Z 702.046,A -85,B 0,C 180,E1 26694.801,E2 26694.801} C_VEL
LIN {X 0,Y 560.425,Z 690.324,A -85,B 0,C 180,E1 26693.553,E2 26693.553} C_VEL
LIN {X 0,Y 560.644,Z 677.033,A -85,B 0,C 180,E1 26692.418,E2 26692.418} C_VEL
LIN {X 0,Y 560.868,Z 662.899,A -85,B 0,C 180,E1 26691.469,E2 26691.469} C_VEL
LIN {X 0,Y 561.089,Z 648.335,A -85,B 0,C 180,E1 26690.708,E2 26690.708} C_VEL
LIN {X 0,Y 561.289,Z 632.212,A -85,B 0,C 180,E1 26690.09,E2 26690.09} C_VEL
LIN {X 0,Y 561.405,Z 615.816,A -85,B 0,C 180,E1 26689.67,E2 26689.67} C_VEL
LIN {X 0,Y 561.631,Z 540.614,A -85,B 0,C 180,E1 26688.668,E2 26688.668} C_VEL
LIN {X 0,Y 561.621,Z 475.594,A -85,B 0,C 180,E1 26687.817,E2 26687.817} C_VEL
LIN {X 0,Y 561.244,Z 472.411,A -85,B 0,C 180,E1 26687.751,E2 26687.751} C_VEL
LIN {X 0,Y 561.705,Z 433.531,A -85,B 0,C 180,E1 26684.822,E2 26684.822} C_VEL
LIN {X 0,Y 562.301,Z 390.839,A -85,B 0,C 180,E1 26681.533,E2 26681.533} C_VEL
LIN {X 0,Y 562.735,Z 360.838,A -85,B 0,C 180,E1 26679.227,E2 26679.227} C_VEL
LIN {X 0,Y 562.922,Z 318.216,A -85,B 0,C 180,E1 26676.01,E2 26676.01} C_VEL
LIN {X 0,Y 562.881,Z 280.091,A -85,B 0,C 180,E1 26673.109,E2 26673.109} C_VEL
LIN {X 0,Y 562.592,Z 274.842,A -85,B 0,C 180,E1 26672.703,E2 26672.703} C_VEL
LIN {X 0,Y 560.307,Z 267.002,A -85,B 0,C 180,E1 26671.975,E2 26671.975} C_VEL
LIN {X 0,Y 560.264,Z 266.699,A -85,B 0,C 180,E1 26671.168,E2 26671.168} C_VEL
LIN {X 0,Y 560.268,Z 266.7,A -85,B 0,C 180,E1 26667.877,E2 26667.877} C_VEL
LIN {X 0,Y 560.234,Z 266.697,A -85,B 0,C 180,E1 26664.573,E2 26664.573} C_VEL
LIN {X 0,Y 560.282,Z 266.692,A -85,B 0,C 180,E1 26661.329,E2 26661.329} C_VEL
LIN {X 0,Y 560.246,Z 266.695,A -85,B 0,C 180,E1 26658.092,E2 26658.092} C_VEL
LIN {X 0,Y 560.241,Z 266.693,A -85,B 0,C 180,E1 26654.681,E2 26654.681} C_VEL
LIN {X 0,Y 560.282,Z 266.695,A -85,B 0,C 180,E1 26651.425,E2 26651.425} C_VEL
LIN {X 0,Y 560.238,Z 266.695,A -85,B 0,C 180,E1 26648.209,E2 26648.209} C_VEL
LIN {X 0,Y 560.268,Z 266.691,A -85,B 0,C 180,E1 26644.914,E2 26644.914} C_VEL
LIN {X 0,Y 560.272,Z 266.698,A -85,B 0,C 180,E1 26641.637,E2 26641.637} C_VEL
LIN {X 0,Y 560.24,Z 266.693,A -85,B 0,C 180,E1 26638.364,E2 26638.364} C_VEL
LIN {X 0,Y 560.283,Z 266.692,A -85,B 0,C 180,E1 26635.086,E2 26635.086} C_VEL
LIN {X 0,Y 560.251,Z 266.697,A -85,B 0,C 180,E1 26631.792,E2 26631.792} C_VEL
LIN {X 0,Y 560.248,Z 266.692,A -85,B 0,C 180,E1 26628.45,E2 26628.45} C_VEL
LIN {X 0,Y 560.281,Z 266.694,A -85,B 0,C 180,E1 26625.215,E2 26625.215} C_VEL
LIN {X 0,Y 560.245,Z 266.695,A -85,B 0,C 180,E1 26621.909,E2 26621.909} C_VEL
LIN {X 0,Y 560.262,Z 266.69,A -85,B 0,C 180,E1 26618.541,E2 26618.541} C_VEL
LIN {X 0,Y 560.283,Z 266.697,A -85,B 0,C 180,E1 26615.205,E2 26615.205} C_VEL
LIN {X 0,Y 560.244,Z 266.694,A -85,B 0,C 180,E1 26611.891,E2 26611.891} C_VEL
LIN {X 0,Y 560.272,Z 266.69,A -85,B 0,C 180,E1 26608.54,E2 26608.54} C_VEL
LIN {X 0,Y 560.278,Z 266.698,A -85,B 0,C 180,E1 26605.172,E2 26605.172} C_VEL
LIN {X 0,Y 560.245,Z 266.694,A -85,B 0,C 180,E1 26601.867,E2 26601.867} C_VEL
LIN {X 0,Y 560.28,Z 266.691,A -85,B 0,C 180,E1 26598.542,E2 26598.542} C_VEL
LIN {X 0,Y 560.278,Z 266.698,A -85,B 0,C 180,E1 26595.178,E2 26595.178} C_VEL
LIN {X 0,Y 560.247,Z 266.695,A -85,B 0,C 180,E1 26591.87,E2 26591.87} C_VEL
LIN {X 0,Y 560.282,Z 266.694,A -85,B 0,C 180,E1 26588.59,E2 26588.59} C_VEL
LIN {X 0,Y 560.268,Z 266.669,A -85,B 0,C 180,E1 26585.198,E2 26585.198} C_VEL
LIN {X 0,Y 560.278,Z 266.906,A -85,B 0,C 180,E1 26583.771,E2 26583.771} C_VEL
LIN {X 0,Y 561.758,Z 271.085,A -85,B 0,C 180,E1 26583.317,E2 26583.317} C_VEL
LIN {X 0,Y 565.073,Z 279.818,A -85,B 0,C 180,E1 26582.473,E2 26582.473} C_VEL
LIN {X 0,Y 564.444,Z 315.729,A -85,B 0,C 180,E1 26580.023,E2 26580.023} C_VEL
LIN {X 0,Y 565.686,Z 324.502,A -85,B 0,C 180,E1 26579.821,E2 26579.821} C_VEL
LIN {X 0,Y 564.555,Z 553.958,A -85,B 0,C 180,E1 26576.64,E2 26576.64} C_VEL
LIN {X 0,Y 564.325,Z 581.698,A -85,B 0,C 180,E1 26576.205,E2 26576.205} C_VEL
LIN {X 0,Y 564.036,Z 601.947,A -85,B 0,C 180,E1 26575.701,E2 26575.701} C_VEL
LIN {X 0,Y 563.663,Z 621.652,A -85,B 0,C 180,E1 26575.021,E2 26575.021} C_VEL
LIN {X 0,Y 563.193,Z 640.59,A -85,B 0,C 180,E1 26574.175,E2 26574.175} C_VEL
LIN {X 0,Y 562.703,Z 659.659,A -85,B 0,C 180,E1 26573.121,E2 26573.121} C_VEL
LIN {X 0,Y 562.187,Z 678.21,A -85,B 0,C 180,E1 26571.874,E2 26571.874} C_VEL
LIN {X 0,Y 561.687,Z 695.631,A -85,B 0,C 180,E1 26570.473,E2 26570.473} C_VEL
LIN {X 0,Y 561.246,Z 711.43,A -85,B 0,C 180,E1 26568.972,E2 26568.972} C_VEL
LIN {X 0,Y 560.855,Z 726.217,A -85,B 0,C 180,E1 26567.319,E2 26567.319} C_VEL
LIN {X 0,Y 560.539,Z 739.871,A -85,B 0,C 180,E1 26565.518,E2 26565.518} C_VEL
LIN {X 0,Y 560.285,Z 751.932,A -85,B 0,C 180,E1 26563.623,E2 26563.623} C_VEL
LIN {X 0,Y 560.111,Z 762.401,A -85,B 0,C 180,E1 26561.636,E2 26561.636} C_VEL
LIN {X 0,Y 560.008,Z 770.879,A -85,B 0,C 180,E1 26559.66,E2 26559.66} C_VEL
LIN {X 0,Y 559.947,Z 777.903,A -85,B 0,C 180,E1 26557.592,E2 26557.592} C_VEL
LIN {X 0,Y 559.916,Z 783.145,A -85,B 0,C 180,E1 26555.532,E2 26555.532} C_VEL
LIN {X 0,Y 559.903,Z 786.711,A -85,B 0,C 180,E1 26553.48,E2 26553.48} C_VEL
LIN {X 0,Y 559.9,Z 788.575,A -85,B 0,C 180,E1 26551.431,E2 26551.431} C_VEL
LIN {X 0,Y 559.901,Z 788.873,A -85,B 0,C 180,E1 26549.385,E2 26549.385} C_VEL
LIN {X 0,Y 559.911,Z 787.504,A -85,B 0,C 180,E1 26547.235,E2 26547.235} C_VEL
LIN {X 0,Y 559.92,Z 784.519,A -85,B 0,C 180,E1 26545.155,E2 26545.155} C_VEL
LIN {X 0,Y 559.936,Z 779.972,A -85,B 0,C 180,E1 26543.128,E2 26543.128} C_VEL
LIN {X 0,Y 559.976,Z 773.909,A -85,B 0,C 180,E1 26541.166,E2 26541.166} C_VEL
LIN {X 0,Y 560.054,Z 766.176,A -85,B 0,C 180,E1 26539.195,E2 26539.195} C_VEL
LIN {X 0,Y 560.192,Z 757.134,A -85,B 0,C 180,E1 26537.317,E2 26537.317} C_VEL
LIN {X 0,Y 560.409,Z 746.174,A -85,B 0,C 180,E1 26535.429,E2 26535.429} C_VEL
LIN {X 0,Y 560.68,Z 733.606,A -85,B 0,C 180,E1 26533.619,E2 26533.619} C_VEL
LIN {X 0,Y 561.017,Z 719.806,A -85,B 0,C 180,E1 26531.933,E2 26531.933} C_VEL
LIN {X 0,Y 561.417,Z 705.224,A -85,B 0,C 180,E1 26530.411,E2 26530.411} C_VEL
LIN {X 0,Y 561.906,Z 687.948,A -85,B 0,C 180,E1 26528.879,E2 26528.879} C_VEL
LIN {X 0,Y 562.422,Z 669.746,A -85,B 0,C 180,E1 26527.528,E2 26527.528} C_VEL
LIN {X 0,Y 562.917,Z 651.36,A -85,B 0,C 180,E1 26526.393,E2 26526.393} C_VEL
LIN {X 0,Y 563.397,Z 633.055,A -85,B 0,C 180,E1 26525.462,E2 26525.462} C_VEL
LIN {X 0,Y 563.826,Z 613.331,A -85,B 0,C 180,E1 26524.67,E2 26524.67} C_VEL
LIN {X 0,Y 564.155,Z 593.353,A -85,B 0,C 180,E1 26524.063,E2 26524.063} C_VEL
LIN {X 0,Y 564.441,Z 572.22,A -85,B 0,C 180,E1 26523.623,E2 26523.623} C_VEL
LIN {X 0,Y 565.636,Z 334.299,A -85,B 0,C 180,E1 26520.316,E2 26520.316} C_VEL
LIN {X 0,Y 565.47,Z 321.725,A -85,B 0,C 180,E1 26520.127,E2 26520.127} C_VEL
LIN {X 0,Y 564.376,Z 315.078,A -85,B 0,C 180,E1 26519.953,E2 26519.953} C_VEL
LIN {X 0,Y 565.074,Z 279.781,A -85,B 0,C 180,E1 26517.524,E2 26517.524} C_VEL
LIN {X 0,Y 560.299,Z 267.044,A -85,B 0,C 180,E1 26516.261,E2 26516.261} C_VEL
LIN {X 0,Y 560.281,Z 266.696,A -85,B 0,C 180,E1 26515.534,E2 26515.534} C_VEL
LIN {X 0,Y 560.243,Z 266.698,A -85,B 0,C 180,E1 26512.243,E2 26512.243} C_VEL
LIN {X 0,Y 560.28,Z 266.699,A -85,B 0,C 180,E1 26508.949,E2 26508.949} C_VEL
LIN {X 0,Y 560.273,Z 266.693,A -85,B 0,C 180,E1 26505.607,E2 26505.607} C_VEL
LIN {X 0,Y 560.238,Z 266.697,A -85,B 0,C 180,E1 26502.286,E2 26502.286} C_VEL
LIN {X 0,Y 560.285,Z 266.697,A -85,B 0,C 180,E1 26499.046,E2 26499.046} C_VEL
LIN {X 0,Y 560.242,Z 266.697,A -85,B 0,C 180,E1 26495.829,E2 26495.829} C_VEL
LIN {X 0,Y 560.235,Z 266.702,A -85,B 0,C 180,E1 26492.416,E2 26492.416} C_VEL
LIN {X 0,Y 560.316,Z 266.965,A -85,B 0,C 180,E1 26491.343,E2 26491.343} C_VEL
LIN {X 0,Y 563.994,Z 278.837,A -85,B 0,C 180,E1 26490.113,E2 26490.113} C_VEL
LIN {X 0,Y 563.168,Z 320.602,A -85,B 0,C 180,E1 26486.805,E2 26486.805} C_VEL
LIN {X 0,Y 562.846,Z 342.314,A -85,B 0,C 180,E1 26485.137,E2 26485.137} C_VEL
LIN {X 0,Y 564.008,Z 350.714,A -85,B 0,C 180,E1 26484.952,E2 26484.952} C_VEL
LIN {X 0,Y 563.116,Z 559.798,A -85,B 0,C 180,E1 26482.115,E2 26482.115} C_VEL
LIN {X 0,Y 562.874,Z 579.546,A -85,B 0,C 180,E1 26481.649,E2 26481.649} C_VEL
LIN {X 0,Y 562.57,Z 598.215,A -85,B 0,C 180,E1 26481.012,E2 26481.012} C_VEL
LIN {X 0,Y 562.198,Z 616.486,A -85,B 0,C 180,E1 26480.183,E2 26480.183} C_VEL
LIN {X 0,Y 561.806,Z 634.182,A -85,B 0,C 180,E1 26479.169,E2 26479.169} C_VEL
LIN {X 0,Y 561.413,Z 650.716,A -85,B 0,C 180,E1 26478.002,E2 26478.002} C_VEL
LIN {X 0,Y 561.036,Z 666.26,A -85,B 0,C 180,E1 26476.674,E2 26476.674} C_VEL
LIN {X 0,Y 560.702,Z 680.641,A -85,B 0,C 180,E1 26475.196,E2 26475.196} C_VEL
LIN {X 0,Y 560.439,Z 693.485,A -85,B 0,C 180,E1 26473.621,E2 26473.621} C_VEL
LIN {X 0,Y 560.226,Z 704.816,A -85,B 0,C 180,E1 26471.948,E2 26471.948} C_VEL
LIN {X 0,Y 560.085,Z 714.653,A -85,B 0,C 180,E1 26470.179,E2 26470.179} C_VEL
LIN {X 0,Y 559.984,Z 722.97,A -85,B 0,C 180,E1 26468.315,E2 26468.315} C_VEL
LIN {X 0,Y 559.938,Z 729.715,A -85,B 0,C 180,E1 26466.356,E2 26466.356} C_VEL
LIN {X 0,Y 559.912,Z 734.545,A -85,B 0,C 180,E1 26464.404,E2 26464.404} C_VEL
